	W =  90.000 deg,	P =   0.000 deg,	R =   90.000 deg
};
P[960]{
   GP1:
	UF : 0, UT : 6,		CONFIG : 'N U T, 0, 0, 0',
	X =  -28.903  mm,	Y =   -328.878  mm,	Z =   -247.975  mm,
	W =  90.000 deg,	P =   0.000 deg,	R =   90.000 deg
};
P[961]{
   GP1:
	UF : 0, UT : 6,		CONFIG : 'N U T, 0, 0, 0',
	X =  -30.345  mm,	Y =   -329.747  mm,	Z =   -248.064  mm,
	W =  90.000 deg,	P =   0.000 deg,	R =   90.000 deg
};
P[962]{
   GP1:
	UF : 0, UT : 6,		CONFIG : 'N U T, 0, 0, 0',
	X =  -31.296  mm,	Y =   -330.198  mm,	Z =   -247.828  mm,
	W =  90.000 deg,	P =   0.000 deg,	R =   90.000 deg
};
P[963]{
   GP1:
	UF : 0, UT : 6,		CONFIG : 'N U T, 0, 0, 0',
	X =  -37.082  mm,	Y =   -333.556  mm,	Z =   -247.870  mm,
	W =  90.000 deg,	P =   0.000 deg,	R =   90.000 deg
};
P[964]{
   GP1:
	UF : 0, UT : 6,		CONFIG : 'N U T, 0, 0, 0',
	X =  -38.322  mm,	Y =   -334.338  mm,	Z =   -248.027  mm,
	W =  90.000 deg,	P =   0.000 deg,	R =   90.000 deg
};
P[965]{
   GP1:
	UF : 0, UT : 6,		CONFIG : 'N U T, 0, 0, 0',
	X =  -39.006  mm,	Y =   -334.749  mm,	Z =   -248.069  mm,
	W =  90.000 deg,	P =   0.000 deg,	R =   90.000 deg
};
P[966]{
   GP1:
	UF : 0, UT : 6,		CONFIG : 'N U T, 0, 0, 0',
	X =  -40.131  mm,	Y =   -335.448  mm,	Z =   -248.189  mm,
	W =  90.000 deg,	P =   0.000 deg,	R =   90.000 deg
};
P[967]{
   GP1:
	UF : 0, UT : 6,		CONFIG : 'N U T, 0, 0, 0',
	X =  -41.021  mm,	Y =   -335.924  mm,	Z =   -248.096  mm,
	W =  90.000 deg,	P =   0.000 deg,	R =   90.000 deg
};
P[968]{
   GP1:
	UF : 0, UT : 6,		CONFIG : 'N U T, 0, 0, 0',
	X =  -42.003  mm,	Y =   -336.481  mm,	Z =   -248.073  mm,
	W =  90.000 deg,	P =   0.000 deg,	R =   90.000 deg
};
P[969]{
   GP1:
	UF : 0, UT : 6,		CONFIG : 'N U T, 0, 0, 0',
	X =  -43.049  mm,	Y =   -337.147  mm,	Z =   -248.222  mm,
	W =  90.000 deg,	P =   0.000 deg,	R =   90.000 deg
};
P[970]{
   GP1:
	UF : 0, UT : 6,		CONFIG : 'N U T, 0, 0, 0',
	X =  -43.885  mm,	Y =   -337.634  mm,	Z =   -248.233  mm,
	W =  90.000 deg,	P =   0.000 deg,	R =   90.000 deg
};
P[971]{
   GP1:
	UF : 0, UT : 6,		CONFIG : 'N U T, 0, 0, 0',
	X =  -45.078  mm,	Y =   -338.309  mm,	Z =   -248.202  mm,
	W =  90.000 deg,	P =   0.000 deg,	R =   90.000 deg
};
P[972]{
   GP1:
	UF : 0, UT : 6,		CONFIG : 'N U T, 0, 0, 0',
	X =  -49.857  mm,	Y =   -340.939  mm,	Z =   -247.886  mm,
	W =  90.000 deg,	P =   0.000 deg,	R =   90.000 deg
};
P[973]{
   GP1:
	UF : 0, UT : 6,		CONFIG : 'N U T, 0, 0, 0',
	X =  -51.596  mm,	Y =   -342.068  mm,	Z =   -248.190  mm,
	W =  90.000 deg,	P =   0.000 deg,	R =   90.000 deg
};
P[974]{
   GP1:
	UF : 0, UT : 6,		CONFIG : 'N U T, 0, 0, 0',
	X =  -55.566  mm,	Y =   -344.197  mm,	Z =   -247.792  mm,
	W =  90.000 deg,	P =   0.000 deg,	R =   90.000 deg
};
P[975]{
   GP1:
	UF : 0, UT : 6,		CONFIG : 'N U T, 0, 0, 0',
	X =  -56.702  mm,	Y =   -344.999  mm,	Z =   -248.147  mm,
	W =  90.000 deg,	P =   0.000 deg,	R =   90.000 deg
};
P[976]{
   GP1:
	UF : 0, UT : 6,		CONFIG : 'N U T, 0, 0, 0',
	X =  -58.375  mm,	Y =   -345.890  mm,	Z =   -247.965  mm,
	W =  90.000 deg,	P =   0.000 deg,	R =   90.000 deg
};
P[977]{
   GP1:
	UF : 0, UT : 6,		CONFIG : 'N U T, 0, 0, 0',
	X =  -60.750  mm,	Y =   -347.335  mm,	Z =   -248.145  mm,
	W =  90.000 deg,	P =   0.000 deg,	R =   90.000 deg
};
P[978]{
   GP1:
	UF : 0, UT : 6,		CONFIG : 'N U T, 0, 0, 0',
	X =  -61.386  mm,	Y =   -347.642  mm,	Z =   -247.998  mm,
	W =  90.000 deg,	P =   0.000 deg,	R =   90.000 deg
};
P[979]{
   GP1:
	UF : 0, UT : 6,		CONFIG : 'N U T, 0, 0, 0',
	X =  -63.196  mm,	Y =   -348.624  mm,	Z =   -247.843  mm,
	W =  90.000 deg,	P =   0.000 deg,	R =   90.000 deg
};
P[980]{
   GP1:
	UF : 0, UT : 6,		CONFIG : 'N U T, 0, 0, 0',
	X =  -64.126  mm,	Y =   -349.230  mm,	Z =   -248.010  mm,
	W =  90.000 deg,	P =   0.000 deg,	R =   90.000 deg
};
P[981]{
   GP1:
	UF : 0, UT : 6,		CONFIG : 'N U T, 0, 0, 0',
	X =  -65.042  mm,	Y =   -349.775  mm,	Z =   -248.050  mm,
	W =  90.000 deg,	P =   0.000 deg,	R =   90.000 deg
};
P[982]{
   GP1:
	UF : 0, UT : 6,		CONFIG : 'N U T, 0, 0, 0',
	X =  -68.055  mm,	Y =   -351.565  mm,	Z =   -248.174  mm,
	W =  90.000 deg,	P =   0.000 deg,	R =   90.000 deg
};
P[983]{
   GP1:
	UF : 0, UT : 6,		CONFIG : 'N U T, 0, 0, 0',
	X =  -70.480  mm,	Y =   -352.838  mm,	Z =   -247.864  mm,
	W =  90.000 deg,	P =   0.000 deg,	R =   90.000 deg
};
P[984]{
   GP1:
	UF : 0, UT : 6,		CONFIG : 'N U T, 0, 0, 0',
	X =  -72.242  mm,	Y =   -353.967  mm,	Z =   -248.135  mm,
	W =  90.000 deg,	P =   0.000 deg,	R =   90.000 deg
};
P[985]{
   GP1:
	UF : 0, UT : 6,		CONFIG : 'N U T, 0, 0, 0',
	X =  -73.253  mm,	Y =   -354.525  mm,	Z =   -248.074  mm,
	W =  90.000 deg,	P =   0.000 deg,	R =   90.000 deg
};
P[986]{
   GP1:
	UF : 0, UT : 6,		CONFIG : 'N U T, 0, 0, 0',
	X =  -74.249  mm,	Y =   -355.111  mm,	Z =   -248.099  mm,
	W =  90.000 deg,	P =   0.000 deg,	R =   90.000 deg
};
P[987]{
   GP1:
	UF : 0, UT : 6,		CONFIG : 'N U T, 0, 0, 0',
	X =  -75.340  mm,	Y =   -355.605  mm,	Z =   -247.770  mm,
	W =  90.000 deg,	P =   0.000 deg,	R =   90.000 deg
};
P[988]{
   GP1:
	UF : 0, UT : 6,		CONFIG : 'N U T, 0, 0, 0',
	X =  -77.108  mm,	Y =   -356.686  mm,	Z =   -247.916  mm,
	W =  90.000 deg,	P =   0.000 deg,	R =   90.000 deg
};
P[989]{
   GP1:
	UF : 0, UT : 6,		CONFIG : 'N U T, 0, 0, 0',
	X =  -77.787  mm,	Y =   -357.064  mm,	Z =   -247.884  mm,
	W =  90.000 deg,	P =   0.000 deg,	R =   90.000 deg
};
P[990]{
   GP1:
	UF : 0, UT : 6,		CONFIG : 'N U T, 0, 0, 0',
	X =  -79.134  mm,	Y =   -357.855  mm,	Z =   -247.913  mm,
	W =  90.000 deg,	P =   0.000 deg,	R =   90.000 deg
};
P[991]{
   GP1:
	UF : 0, UT : 6,		CONFIG : 'N U T, 0, 0, 0',
	X =  -81.215  mm,	Y =   -359.115  mm,	Z =   -248.054  mm,
	W =  90.000 deg,	P =   0.000 deg,	R =   90.000 deg
};
P[992]{
   GP1:
	UF : 0, UT : 6,		CONFIG : 'N U T, 0, 0, 0',
	X =  -82.562  mm,	Y =   -359.948  mm,	Z =   -248.191  mm,
	W =  90.000 deg,	P =   0.000 deg,	R =   90.000 deg
};
P[993]{
   GP1:
	UF : 0, UT : 6,		CONFIG : 'N U T, 0, 0, 0',
	X =  -84.553  mm,	Y =   -361.046  mm,	Z =   -248.064  mm,
	W =  90.000 deg,	P =   0.000 deg,	R =   90.000 deg
};
P[994]{
   GP1:
	UF : 0, UT : 6,		CONFIG : 'N U T, 0, 0, 0',
	X =  -85.474  mm,	Y =   -361.519  mm,	Z =   -247.920  mm,
	W =  90.000 deg,	P =   0.000 deg,	R =   90.000 deg
};
P[995]{
   GP1:
	UF : 0, UT : 6,		CONFIG : 'N U T, 0, 0, 0',
	X =  -86.598  mm,	Y =   -362.225  mm,	Z =   -248.060  mm,
	W =  90.000 deg,	P =   0.000 deg,	R =   90.000 deg
};
P[996]{
   GP1:
	UF : 0, UT : 6,		CONFIG : 'N U T, 0, 0, 0',
	X =  -89.940  mm,	Y =   -364.214  mm,	Z =   -248.203  mm,
	W =  90.000 deg,	P =   0.000 deg,	R =   90.000 deg
};
P[997]{
   GP1:
	UF : 0, UT : 6,		CONFIG : 'N U T, 0, 0, 0',
	X =  -90.933  mm,	Y =   -364.603  mm,	Z =   -247.758  mm,
	W =  90.000 deg,	P =   0.000 deg,	R =   90.000 deg
};
P[998]{
   GP1:
	UF : 0, UT : 6,		CONFIG : 'N U T, 0, 0, 0',
	X =  -91.875  mm,	Y =   -365.326  mm,	Z =   -248.193  mm,
	W =  90.000 deg,	P =   0.000 deg,	R =   90.000 deg
};
P[999]{
   GP1:
	UF : 0, UT : 6,		CONFIG : 'N U T, 0, 0, 0',
	X =  -94.257  mm,	Y =   -366.581  mm,	Z =   -247.899  mm,
	W =  90.000 deg,	P =   0.000 deg,	R =   90.000 deg
};
P[1000]{
   GP1:
	UF : 0, UT : 6,		CONFIG : 'N U T, 0, 0, 0',
	X =  -95.224  mm,	Y =   -367.210  mm,	Z =   -248.072  mm,
	W =  90.000 deg,	P =   0.000 deg,	R =   90.000 deg
};
P[1001]{
   GP1:
	UF : 0, UT : 6,		CONFIG : 'N U T, 0, 0, 0',
	X =  -96.301  mm,	Y =   -367.796  mm,	Z =   -247.984  mm,
	W =  90.000 deg,	P =   0.000 deg,	R =   90.000 deg
};
P[1002]{
   GP1:
	UF : 0, UT : 6,		CONFIG : 'N U T, 0, 0, 0',
	X =  -97.537  mm,	Y =   -368.595  mm,	Z =   -248.191  mm,
	W =  90.000 deg,	P =   0.000 deg,	R =   90.000 deg
};
P[1003]{
   GP1:
	UF : 0, UT : 6,		CONFIG : 'N U T, 0, 0, 0',
	X =  -99.221  mm,	Y =   -369.495  mm,	Z =   -248.013  mm,
	W =  90.000 deg,	P =   0.000 deg,	R =   90.000 deg
};
P[1004]{
   GP1:
	UF : 0, UT : 6,		CONFIG : 'N U T, 0, 0, 0',
	X =  -101.503  mm,	Y =   -370.901  mm,	Z =   -248.231  mm,
	W =  90.000 deg,	P =   0.000 deg,	R =   90.000 deg
};
P[1005]{
   GP1:
	UF : 0, UT : 6,		CONFIG : 'N U T, 0, 0, 0',
	X =  -102.830  mm,	Y =   -371.582  mm,	Z =   -248.024  mm,
	W =  90.000 deg,	P =   0.000 deg,	R =   90.000 deg
};
P[1006]{
   GP1:
	UF : 0, UT : 6,		CONFIG : 'N U T, 0, 0, 0',
	X =  -103.563  mm,	Y =   -371.971  mm,	Z =   -247.940  mm,
	W =  90.000 deg,	P =   0.000 deg,	R =   90.000 deg
};
P[1007]{
   GP1:
	UF : 0, UT : 6,		CONFIG : 'N U T, 0, 0, 0',
	X =  -106.169  mm,	Y =   -373.484  mm,	Z =   -247.960  mm,
	W =  90.000 deg,	P =   0.000 deg,	R =   90.000 deg
};
P[1008]{
   GP1:
	UF : 0, UT : 6,		CONFIG : 'N U T, 0, 0, 0',
	X =  -106.807  mm,	Y =   -373.966  mm,	Z =   -248.237  mm,
	W =  90.000 deg,	P =   0.000 deg,	R =   90.000 deg
};
P[1009]{
   GP1:
	UF : 0, UT : 6,		CONFIG : 'N U T, 0, 0, 0',
	X =  -107.493  mm,	Y =   -374.305  mm,	Z =   -248.100  mm,
	W =  90.000 deg,	P =   0.000 deg,	R =   90.000 deg
};
P[1010]{
   GP1:
	UF : 0, UT : 6,		CONFIG : 'N U T, 0, 0, 0',
	X =  -108.733  mm,	Y =   -375.067  mm,	Z =   -248.210  mm,
	W =  90.000 deg,	P =   0.000 deg,	R =   90.000 deg
};
P[1011]{
   GP1:
	UF : 0, UT : 6,		CONFIG : 'N U T, 0, 0, 0',
	X =  -110.528  mm,	Y =   -376.015  mm,	Z =   -247.997  mm,
	W =  90.000 deg,	P =   0.000 deg,	R =   90.000 deg
};
P[1012]{
   GP1:
	UF : 0, UT : 6,		CONFIG : 'N U T, 0, 0, 0',
	X =  -111.099  mm,	Y =   -376.423  mm,	Z =   -248.185  mm,
	W =  90.000 deg,	P =   0.000 deg,	R =   90.000 deg
};
P[1013]{
   GP1:
	UF : 0, UT : 6,		CONFIG : 'N U T, 0, 0, 0',
	X =  -112.870  mm,	Y =   -377.351  mm,	Z =   -247.957  mm,
	W =  90.000 deg,	P =   0.000 deg,	R =   90.000 deg
};
P[1014]{
   GP1:
	UF : 0, UT : 6,		CONFIG : 'N U T, 0, 0, 0',
	X =  -113.558  mm,	Y =   -377.684  mm,	Z =   -247.799  mm,
	W =  90.000 deg,	P =   0.000 deg,	R =   90.000 deg
};
P[1015]{
   GP1:
	UF : 0, UT : 6,		CONFIG : 'N U T, 0, 0, 0',
	X =  -115.265  mm,	Y =   -378.664  mm,	Z =   -247.786  mm,
	W =  90.000 deg,	P =   0.000 deg,	R =   90.000 deg
};
P[1016]{
   GP1:
	UF : 0, UT : 6,		CONFIG : 'N U T, 0, 0, 0',
	X =  -116.104  mm,	Y =   -379.315  mm,	Z =   -248.189  mm,
	W =  90.000 deg,	P =   0.000 deg,	R =   90.000 deg
};
P[1017]{
   GP1:
	UF : 0, UT : 6,		CONFIG : 'N U T, 0, 0, 0',
	X =  -117.677  mm,	Y =   -380.092  mm,	Z =   -247.871  mm,
	W =  90.000 deg,	P =   0.000 deg,	R =   90.000 deg
};
P[1018]{
   GP1:
	UF : 0, UT : 6,		CONFIG : 'N U T, 0, 0, 0',
	X =  -118.616  mm,	Y =   -380.734  mm,	Z =   -248.113  mm,
	W =  90.000 deg,	P =   0.000 deg,	R =   90.000 deg
};
P[1019]{
   GP1:
	UF : 0, UT : 6,		CONFIG : 'N U T, 0, 0, 0',
	X =  -122.113  mm,	Y =   -382.775  mm,	Z =   -248.168  mm,
	W =  90.000 deg,	P =   0.000 deg,	R =   90.000 deg
};
P[1020]{
   GP1:
	UF : 0, UT : 6,		CONFIG : 'N U T, 0, 0, 0',
	X =  -124.559  mm,	Y =   -384.127  mm,	Z =   -248.019  mm,
	W =  90.000 deg,	P =   0.000 deg,	R =   90.000 deg
};
P[1021]{
   GP1:
	UF : 0, UT : 6,		CONFIG : 'N U T, 0, 0, 0',
	X =  -125.422  mm,	Y =   -384.715  mm,	Z =   -248.238  mm,
	W =  90.000 deg,	P =   0.000 deg,	R =   90.000 deg
};
P[1022]{
   GP1:
	UF : 0, UT : 6,		CONFIG : 'N U T, 0, 0, 0',
	X =  -126.709  mm,	Y =   -385.433  mm,	Z =   -248.142  mm,
	W =  90.000 deg,	P =   0.000 deg,	R =   90.000 deg
};
P[1023]{
   GP1:
	UF : 0, UT : 6,		CONFIG : 'N U T, 0, 0, 0',
	X =  -129.563  mm,	Y =   -387.669  mm,	Z =   -248.167  mm,
	W =  90.000 deg,	P =   0.000 deg,	R =   90.000 deg
};
P[1024]{
   GP1:
	UF : 0, UT : 6,		CONFIG : 'N U T, 0, 0, 0',
	X =  -130.198  mm,	Y =   -388.316  mm,	Z =   -248.069  mm,
	W =  90.000 deg,	P =   0.000 deg,	R =   90.000 deg
};
P[1025]{
   GP1:
	UF : 0, UT : 6,		CONFIG : 'N U T, 0, 0, 0',
	X =  -132.423  mm,	Y =   -391.705  mm,	Z =   -248.118  mm,
	W =  90.000 deg,	P =   0.000 deg,	R =   90.000 deg
};
P[1026]{
   GP1:
	UF : 0, UT : 6,		CONFIG : 'N U T, 0, 0, 0',
	X =  -132.726  mm,	Y =   -392.586  mm,	Z =   -248.245  mm,
	W =  90.000 deg,	P =   0.000 deg,	R =   90.000 deg
};
P[1027]{
   GP1:
	UF : 0, UT : 6,		CONFIG : 'N U T, 0, 0, 0',
	X =  -133.115  mm,	Y =   -393.723  mm,	Z =   -248.116  mm,
	W =  90.000 deg,	P =   0.000 deg,	R =   90.000 deg
};
P[1028]{
   GP1:
	UF : 0, UT : 6,		CONFIG : 'N U T, 0, 0, 0',
	X =  -133.602  mm,	Y =   -396.256  mm,	Z =   -247.992  mm,
	W =  90.000 deg,	P =   0.000 deg,	R =   90.000 deg
};
P[1029]{
   GP1:
	UF : 0, UT : 6,		CONFIG : 'N U T, 0, 0, 0',
	X =  -133.574  mm,	Y =   -398.321  mm,	Z =   -248.077  mm,
	W =  90.000 deg,	P =   0.000 deg,	R =   90.000 deg
};
P[1030]{
   GP1:
	UF : 0, UT : 6,		CONFIG : 'N U T, 0, 0, 0',
	X =  -133.207  mm,	Y =   -400.061  mm,	Z =   -248.179  mm,
	W =  90.000 deg,	P =   0.000 deg,	R =   90.000 deg
};
P[1031]{
   GP1:
	UF : 0, UT : 6,		CONFIG : 'N U T, 0, 0, 0',
	X =  -132.889  mm,	Y =   -401.383  mm,	Z =   -248.224  mm,
	W =  90.000 deg,	P =   0.000 deg,	R =   90.000 deg
};
P[1032]{
   GP1:
	UF : 0, UT : 6,		CONFIG : 'N U T, 0, 0, 0',
	X =  -132.012  mm,	Y =   -403.554  mm,	Z =   -248.053  mm,
	W =  90.000 deg,	P =   0.000 deg,	R =   90.000 deg
};
P[1033]{
   GP1:
	UF : 0, UT : 6,		CONFIG : 'N U T, 0, 0, 0',
	X =  -131.322  mm,	Y =   -404.824  mm,	Z =   -248.139  mm,
	W =  90.000 deg,	P =   0.000 deg,	R =   90.000 deg
};
P[1034]{
   GP1:
	UF : 0, UT : 6,		CONFIG : 'N U T, 0, 0, 0',
	X =  -130.983  mm,	Y =   -405.432  mm,	Z =   -248.111  mm,
	W =  90.000 deg,	P =   0.000 deg,	R =   90.000 deg
};
P[1035]{
   GP1:
	UF : 0, UT : 6,		CONFIG : 'N U T, 0, 0, 0',
	X =  -130.285  mm,	Y =   -406.743  mm,	Z =   -247.966  mm,
	W =  90.000 deg,	P =   0.000 deg,	R =   90.000 deg
};
P[1036]{
   GP1:
	UF : 0, UT : 6,		CONFIG : 'N U T, 0, 0, 0',
	X =  -129.882  mm,	Y =   -407.354  mm,	Z =   -248.089  mm,
	W =  90.000 deg,	P =   0.000 deg,	R =   90.000 deg
};
P[1037]{
   GP1:
	UF : 0, UT : 6,		CONFIG : 'N U T, 0, 0, 0',
	X =  -128.584  mm,	Y =   -409.650  mm,	Z =   -248.021  mm,
	W =  90.000 deg,	P =   0.000 deg,	R =   90.000 deg
};
P[1038]{
   GP1:
	UF : 0, UT : 6,		CONFIG : 'N U T, 0, 0, 0',
	X =  -127.392  mm,	Y =   -411.883  mm,	Z =   -247.787  mm,
	W =  90.000 deg,	P =   0.000 deg,	R =   90.000 deg
};
P[1039]{
   GP1:
	UF : 0, UT : 6,		CONFIG : 'N U T, 0, 0, 0',
	X =  -126.637  mm,	Y =   -412.966  mm,	Z =   -248.099  mm,
	W =  90.000 deg,	P =   0.000 deg,	R =   90.000 deg
};
P[1040]{
   GP1:
	UF : 0, UT : 6,		CONFIG : 'N U T, 0, 0, 0',
	X =  -122.435  mm,	Y =   -420.253  mm,	Z =   -248.085  mm,
	W =  90.000 deg,	P =   0.000 deg,	R =   90.000 deg
};
P[1041]{
   GP1:
	UF : 0, UT : 6,		CONFIG : 'N U T, 0, 0, 0',
	X =  -121.804  mm,	Y =   -421.568  mm,	Z =   -247.775  mm,
	W =  90.000 deg,	P =   0.000 deg,	R =   90.000 deg
};
P[1042]{
   GP1:
	UF : 0, UT : 6,		CONFIG : 'N U T, 0, 0, 0',
	X =  -120.774  mm,	Y =   -423.206  mm,	Z =   -247.982  mm,
	W =  90.000 deg,	P =   0.000 deg,	R =   90.000 deg
};
P[1043]{
   GP1:
	UF : 0, UT : 6,		CONFIG : 'N U T, 0, 0, 0',
	X =  -120.097  mm,	Y =   -424.195  mm,	Z =   -248.237  mm,
	W =  90.000 deg,	P =   0.000 deg,	R =   90.000 deg
};
P[1044]{
   GP1:
	UF : 0, UT : 6,		CONFIG : 'N U T, 0, 0, 0',
	X =  -119.414  mm,	Y =   -425.491  mm,	Z =   -248.078  mm,
	W =  90.000 deg,	P =   0.000 deg,	R =   90.000 deg
};
P[1045]{
   GP1:
	UF : 0, UT : 6,		CONFIG : 'N U T, 0, 0, 0',
	X =  -118.894  mm,	Y =   -426.411  mm,	Z =   -248.052  mm,
	W =  90.000 deg,	P =   0.000 deg,	R =   90.000 deg
};
P[1046]{
   GP1:
	UF : 0, UT : 6,		CONFIG : 'N U T, 0, 0, 0',
	X =  -118.256  mm,	Y =   -427.421  mm,	Z =   -248.184  mm,
	W =  90.000 deg,	P =   0.000 deg,	R =   90.000 deg
};
P[1047]{
   GP1:
	UF : 0, UT : 6,		CONFIG : 'N U T, 0, 0, 0',
	X =  -117.760  mm,	Y =   -428.344  mm,	Z =   -248.095  mm,
	W =  90.000 deg,	P =   0.000 deg,	R =   90.000 deg
};
P[1048]{
   GP1:
	UF : 0, UT : 6,		CONFIG : 'N U T, 0, 0, 0',
	X =  -116.499  mm,	Y =   -430.746  mm,	Z =   -247.790  mm,
	W =  90.000 deg,	P =   0.000 deg,	R =   90.000 deg
};
P[1049]{
   GP1:
	UF : 0, UT : 6,		CONFIG : 'N U T, 0, 0, 0',
	X =  -115.798  mm,	Y =   -431.817  mm,	Z =   -247.989  mm,
	W =  90.000 deg,	P =   0.000 deg,	R =   90.000 deg
};
P[1050]{
   GP1:
	UF : 0, UT : 6,		CONFIG : 'N U T, 0, 0, 0',
	X =  -114.795  mm,	Y =   -433.512  mm,	Z =   -248.050  mm,
	W =  90.000 deg,	P =   0.000 deg,	R =   90.000 deg
};
P[1051]{
   GP1:
	UF : 0, UT : 6,		CONFIG : 'N U T, 0, 0, 0',
	X =  -114.179  mm,	Y =   -434.555  mm,	Z =   -248.082  mm,
	W =  90.000 deg,	P =   0.000 deg,	R =   90.000 deg
};
P[1052]{
   GP1:
	UF : 0, UT : 6,		CONFIG : 'N U T, 0, 0, 0',
	X =  -112.942  mm,	Y =   -436.662  mm,	Z =   -248.134  mm,
	W =  90.000 deg,	P =   0.000 deg,	R =   90.000 deg
};
P[1053]{
   GP1:
	UF : 0, UT : 6,		CONFIG : 'N U T, 0, 0, 0',
	X =  -112.334  mm,	Y =   -437.964  mm,	Z =   -247.783  mm,
	W =  90.000 deg,	P =   0.000 deg,	R =   90.000 deg
};
P[1054]{
   GP1:
	UF : 0, UT : 6,		CONFIG : 'N U T, 0, 0, 0',
	X =  -111.595  mm,	Y =   -439.228  mm,	Z =   -247.806  mm,
	W =  90.000 deg,	P =   0.000 deg,	R =   90.000 deg
};
P[1055]{
   GP1:
	UF : 0, UT : 6,		CONFIG : 'N U T, 0, 0, 0',
	X =  -110.365  mm,	Y =   -441.151  mm,	Z =   -248.096  mm,
	W =  90.000 deg,	P =   0.000 deg,	R =   90.000 deg
};
P[1056]{
   GP1:
	UF : 0, UT : 6,		CONFIG : 'N U T, 0, 0, 0',
	X =  -109.824  mm,	Y =   -442.301  mm,	Z =   -247.797  mm,
	W =  90.000 deg,	P =   0.000 deg,	R =   90.000 deg
};
P[1057]{
   GP1:
	UF : 0, UT : 6,		CONFIG : 'N U T, 0, 0, 0',
	X =  -108.955  mm,	Y =   -443.499  mm,	Z =   -248.227  mm,
	W =  90.000 deg,	P =   0.000 deg,	R =   90.000 deg
};
P[1058]{
   GP1:
	UF : 0, UT : 6,		CONFIG : 'N U T, 0, 0, 0',
	X =  -108.580  mm,	Y =   -444.387  mm,	Z =   -247.895  mm,
	W =  90.000 deg,	P =   0.000 deg,	R =   90.000 deg
};
P[1059]{
   GP1:
	UF : 0, UT : 6,		CONFIG : 'N U T, 0, 0, 0',
	X =  -107.695  mm,	Y =   -445.733  mm,	Z =   -248.155  mm,
	W =  90.000 deg,	P =   0.000 deg,	R =   90.000 deg
};
P[1060]{
   GP1:
	UF : 0, UT : 6,		CONFIG : 'N U T, 0, 0, 0',
	X =  -105.502  mm,	Y =   -449.497  mm,	Z =   -248.203  mm,
	W =  90.000 deg,	P =   0.000 deg,	R =   90.000 deg
};
P[1061]{
   GP1:
	UF : 0, UT : 6,		CONFIG : 'N U T, 0, 0, 0',
	X =  -104.845  mm,	Y =   -450.741  mm,	Z =   -248.054  mm,
	W =  90.000 deg,	P =   0.000 deg,	R =   90.000 deg
};
P[1062]{
   GP1:
	UF : 0, UT : 6,		CONFIG : 'N U T, 0, 0, 0',
	X =  -104.462  mm,	Y =   -451.470  mm,	Z =   -247.962  mm,
	W =  90.000 deg,	P =   0.000 deg,	R =   90.000 deg
};
P[1063]{
   GP1:
	UF : 0, UT : 6,		CONFIG : 'N U T, 0, 0, 0',
	X =  -104.089  mm,	Y =   -452.185  mm,	Z =   -247.868  mm,
	W =  90.000 deg,	P =   0.000 deg,	R =   90.000 deg
};
P[1064]{
   GP1:
	UF : 0, UT : 6,		CONFIG : 'N U T, 0, 0, 0',
	X =  -102.684  mm,	Y =   -454.644  mm,	Z =   -247.831  mm,
	W =  90.000 deg,	P =   0.000 deg,	R =   90.000 deg
};
P[1065]{
   GP1:
	UF : 0, UT : 6,		CONFIG : 'N U T, 0, 0, 0',
	X =  -102.091  mm,	Y =   -455.612  mm,	Z =   -247.912  mm,
	W =  90.000 deg,	P =   0.000 deg,	R =   90.000 deg
};
P[1066]{
   GP1:
	UF : 0, UT : 6,		CONFIG : 'N U T, 0, 0, 0',
	X =  -101.461  mm,	Y =   -456.515  mm,	Z =   -248.175  mm,
	W =  90.000 deg,	P =   0.000 deg,	R =   90.000 deg
};
P[1067]{
   GP1:
	UF : 0, UT : 6,		CONFIG : 'N U T, 0, 0, 0',
	X =  -100.753  mm,	Y =   -457.744  mm,	Z =   -248.173  mm,
	W =  90.000 deg,	P =   0.000 deg,	R =   90.000 deg
};
P[1068]{
   GP1:
	UF : 0, UT : 6,		CONFIG : 'N U T, 0, 0, 0',
	X =  -99.853  mm,	Y =   -459.493  mm,	Z =   -247.904  mm,
	W =  90.000 deg,	P =   0.000 deg,	R =   90.000 deg
};
P[1069]{
   GP1:
	UF : 0, UT : 6,		CONFIG : 'N U T, 0, 0, 0',
	X =  -97.147  mm,	Y =   -463.978  mm,	Z =   -248.189  mm,
	W =  90.000 deg,	P =   0.000 deg,	R =   90.000 deg
};
P[1070]{
   GP1:
	UF : 0, UT : 6,		CONFIG : 'N U T, 0, 0, 0',
	X =  -96.488  mm,	Y =   -465.368  mm,	Z =   -247.838  mm,
	W =  90.000 deg,	P =   0.000 deg,	R =   90.000 deg
};
P[1071]{
   GP1:
	UF : 0, UT : 6,		CONFIG : 'N U T, 0, 0, 0',
	X =  -95.821  mm,	Y =   -466.485  mm,	Z =   -247.895  mm,
	W =  90.000 deg,	P =   0.000 deg,	R =   90.000 deg
};
P[1072]{
   GP1:
	UF : 0, UT : 6,		CONFIG : 'N U T, 0, 0, 0',
	X =  -95.262  mm,	Y =   -467.225  mm,	Z =   -248.213  mm,
	W =  90.000 deg,	P =   0.000 deg,	R =   90.000 deg
};
P[1073]{
   GP1:
	UF : 0, UT : 6,		CONFIG : 'N U T, 0, 0, 0',
	X =  -93.623  mm,	Y =   -470.273  mm,	Z =   -247.917  mm,
	W =  90.000 deg,	P =   0.000 deg,	R =   90.000 deg
};
P[1074]{
   GP1:
	UF : 0, UT : 6,		CONFIG : 'N U T, 0, 0, 0',
	X =  -92.822  mm,	Y =   -471.615  mm,	Z =   -247.983  mm,
	W =  90.000 deg,	P =   0.000 deg,	R =   90.000 deg
};
P[1075]{
   GP1:
	UF : 0, UT : 6,		CONFIG : 'N U T, 0, 0, 0',
	X =  -92.155  mm,	Y =   -472.636  mm,	Z =   -248.172  mm,
	W =  90.000 deg,	P =   0.000 deg,	R =   90.000 deg
};
P[1076]{
   GP1:
	UF : 0, UT : 6,		CONFIG : 'N U T, 0, 0, 0',
	X =  -91.150  mm,	Y =   -474.438  mm,	Z =   -248.086  mm,
	W =  90.000 deg,	P =   0.000 deg,	R =   90.000 deg
};
P[1077]{
   GP1:
	UF : 0, UT : 6,		CONFIG : 'N U T, 0, 0, 0',
	X =  -90.497  mm,	Y =   -475.686  mm,	Z =   -247.922  mm,
	W =  90.000 deg,	P =   0.000 deg,	R =   90.000 deg
};
P[1078]{
   GP1:
	UF : 0, UT : 6,		CONFIG : 'N U T, 0, 0, 0',
	X =  -88.747  mm,	Y =   -478.722  mm,	Z =   -247.912  mm,
	W =  90.000 deg,	P =   0.000 deg,	R =   90.000 deg
};
P[1079]{
   GP1:
	UF : 0, UT : 6,		CONFIG : 'N U T, 0, 0, 0',
	X =  -88.249  mm,	Y =   -479.554  mm,	Z =   -247.957  mm,
	W =  90.000 deg,	P =   0.000 deg,	R =   90.000 deg
};
P[1080]{
   GP1:
	UF : 0, UT : 6,		CONFIG : 'N U T, 0, 0, 0',
	X =  -87.020  mm,	Y =   -481.678  mm,	Z =   -247.963  mm,
	W =  90.000 deg,	P =   0.000 deg,	R =   90.000 deg
};
P[1081]{
   GP1:
	UF : 0, UT : 6,		CONFIG : 'N U T, 0, 0, 0',
	X =  -86.491  mm,	Y =   -482.557  mm,	Z =   -248.017  mm,
	W =  90.000 deg,	P =   0.000 deg,	R =   90.000 deg
};
P[1082]{
   GP1:
	UF : 0, UT : 6,		CONFIG : 'N U T, 0, 0, 0',
	X =  -83.260  mm,	Y =   -488.237  mm,	Z =   -247.897  mm,
	W =  90.000 deg,	P =   0.000 deg,	R =   90.000 deg
};
P[1083]{
   GP1:
	UF : 0, UT : 6,		CONFIG : 'N U T, 0, 0, 0',
	X =  -81.554  mm,	Y =   -491.053  mm,	Z =   -248.092  mm,
	W =  90.000 deg,	P =   0.000 deg,	R =   90.000 deg
};
P[1084]{
   GP1:
	UF : 0, UT : 6,		CONFIG : 'N U T, 0, 0, 0',
	X =  -79.066  mm,	Y =   -495.264  mm,	Z =   -248.227  mm,
	W =  90.000 deg,	P =   0.000 deg,	R =   90.000 deg
};
P[1085]{
   GP1:
	UF : 0, UT : 6,		CONFIG : 'N U T, 0, 0, 0',
	X =  -78.745  mm,	Y =   -496.131  mm,	Z =   -247.793  mm,
	W =  90.000 deg,	P =   0.000 deg,	R =   90.000 deg
};
P[1086]{
   GP1:
	UF : 0, UT : 6,		CONFIG : 'N U T, 0, 0, 0',
	X =  -76.359  mm,	Y =   -499.951  mm,	Z =   -248.231  mm,
	W =  90.000 deg,	P =   0.000 deg,	R =   90.000 deg
};
P[1087]{
   GP1:
	UF : 0, UT : 6,		CONFIG : 'N U T, 0, 0, 0',
	X =  -75.085  mm,	Y =   -502.217  mm,	Z =   -248.147  mm,
	W =  90.000 deg,	P =   0.000 deg,	R =   90.000 deg
};
P[1088]{
   GP1:
	UF : 0, UT : 6,		CONFIG : 'N U T, 0, 0, 0',
	X =  -74.296  mm,	Y =   -503.735  mm,	Z =   -247.934  mm,
	W =  90.000 deg,	P =   0.000 deg,	R =   90.000 deg
};
P[1089]{
   GP1:
	UF : 0, UT : 6,		CONFIG : 'N U T, 0, 0, 0',
	X =  -73.716  mm,	Y =   -504.717  mm,	Z =   -247.965  mm,
	W =  90.000 deg,	P =   0.000 deg,	R =   90.000 deg
};
P[1090]{
   GP1:
	UF : 0, UT : 6,		CONFIG : 'N U T, 0, 0, 0',
	X =  -73.101  mm,	Y =   -505.743  mm,	Z =   -248.019  mm,
	W =  90.000 deg,	P =   0.000 deg,	R =   90.000 deg
};
P[1091]{
   GP1:
	UF : 0, UT : 6,		CONFIG : 'N U T, 0, 0, 0',
	X =  -72.668  mm,	Y =   -506.616  mm,	Z =   -247.847  mm,
	W =  90.000 deg,	P =   0.000 deg,	R =   90.000 deg
};
P[1092]{
   GP1:
	UF : 0, UT : 6,		CONFIG : 'N U T, 0, 0, 0',
	X =  -71.102  mm,	Y =   -509.080  mm,	Z =   -248.194  mm,
	W =  90.000 deg,	P =   0.000 deg,	R =   90.000 deg
};
P[1093]{
   GP1:
	UF : 0, UT : 6,		CONFIG : 'N U T, 0, 0, 0',
	X =  -69.772  mm,	Y =   -511.607  mm,	Z =   -247.882  mm,
	W =  90.000 deg,	P =   0.000 deg,	R =   90.000 deg
};
P[1094]{
   GP1:
	UF : 0, UT : 6,		CONFIG : 'N U T, 0, 0, 0',
	X =  -68.834  mm,	Y =   -513.104  mm,	Z =   -248.060  mm,
	W =  90.000 deg,	P =   0.000 deg,	R =   90.000 deg
};
P[1095]{
   GP1:
	UF : 0, UT : 6,		CONFIG : 'N U T, 0, 0, 0',
	X =  -68.421  mm,	Y =   -513.798  mm,	Z =   -248.091  mm,
	W =  90.000 deg,	P =   0.000 deg,	R =   90.000 deg
};
P[1096]{
   GP1:
	UF : 0, UT : 6,		CONFIG : 'N U T, 0, 0, 0',
	X =  -67.867  mm,	Y =   -514.903  mm,	Z =   -247.889  mm,
	W =  90.000 deg,	P =   0.000 deg,	R =   90.000 deg
};
P[1097]{
   GP1:
	UF : 0, UT : 6,		CONFIG : 'N U T, 0, 0, 0',
	X =  -67.447  mm,	Y =   -515.576  mm,	Z =   -247.964  mm,
	W =  90.000 deg,	P =   0.000 deg,	R =   90.000 deg
};
P[1098]{
   GP1:
	UF : 0, UT : 6,		CONFIG : 'N U T, 0, 0, 0',
	X =  -65.365  mm,	Y =   -519.077  mm,	Z =   -248.110  mm,
	W =  90.000 deg,	P =   0.000 deg,	R =   90.000 deg
};
P[1099]{
   GP1:
	UF : 0, UT : 6,		CONFIG : 'N U T, 0, 0, 0',
	X =  -64.641  mm,	Y =   -520.439  mm,	Z =   -247.960  mm,
	W =  90.000 deg,	P =   0.000 deg,	R =   90.000 deg
};
P[1100]{
   GP1:
	UF : 0, UT : 6,		CONFIG : 'N U T, 0, 0, 0',
	X =  -63.019  mm,	Y =   -523.252  mm,	Z =   -247.954  mm,
	W =  90.000 deg,	P =   0.000 deg,	R =   90.000 deg
};
P[1101]{
   GP1:
	UF : 0, UT : 6,		CONFIG : 'N U T, 0, 0, 0',
	X =  -61.572  mm,	Y =   -525.772  mm,	Z =   -247.935  mm,
	W =  90.000 deg,	P =   0.000 deg,	R =   90.000 deg
};
P[1102]{
   GP1:
	UF : 0, UT : 6,		CONFIG : 'N U T, 0, 0, 0',
	X =  -57.398  mm,	Y =   -532.795  mm,	Z =   -248.222  mm,
	W =  90.000 deg,	P =   0.000 deg,	R =   90.000 deg
};
P[1103]{
   GP1:
	UF : 0, UT : 6,		CONFIG : 'N U T, 0, 0, 0',
	X =  -56.956  mm,	Y =   -533.648  mm,	Z =   -248.101  mm,
	W =  90.000 deg,	P =   0.000 deg,	R =   90.000 deg
};
P[1104]{
   GP1:
	UF : 0, UT : 6,		CONFIG : 'N U T, 0, 0, 0',
	X =  -53.366  mm,	Y =   -539.846  mm,	Z =   -248.130  mm,
	W =  90.000 deg,	P =   0.000 deg,	R =   90.000 deg
};
P[1105]{
   GP1:
	UF : 0, UT : 6,		CONFIG : 'N U T, 0, 0, 0',
	X =  -52.923  mm,	Y =   -540.786  mm,	Z =   -247.884  mm,
	W =  90.000 deg,	P =   0.000 deg,	R =   90.000 deg
};
P[1106]{
   GP1:
	UF : 0, UT : 6,		CONFIG : 'N U T, 0, 0, 0',
	X =  -52.193  mm,	Y =   -542.081  mm,	Z =   -247.845  mm,
	W =  90.000 deg,	P =   0.000 deg,	R =   90.000 deg
};
P[1107]{
   GP1:
	UF : 0, UT : 6,		CONFIG : 'N U T, 0, 0, 0',
	X =  -50.214  mm,	Y =   -545.475  mm,	Z =   -247.891  mm,
	W =  90.000 deg,	P =   0.000 deg,	R =   90.000 deg
};
P[1108]{
   GP1:
	UF : 0, UT : 6,		CONFIG : 'N U T, 0, 0, 0',
	X =  -49.708  mm,	Y =   -546.190  mm,	Z =   -248.114  mm,
	W =  90.000 deg,	P =   0.000 deg,	R =   90.000 deg
};
P[1109]{
   GP1:
	UF : 0, UT : 6,		CONFIG : 'N U T, 0, 0, 0',
	X =  -49.193  mm,	Y =   -547.125  mm,	Z =   -248.057  mm,
	W =  90.000 deg,	P =   0.000 deg,	R =   90.000 deg
};
P[1110]{
   GP1:
	UF : 0, UT : 6,		CONFIG : 'N U T, 0, 0, 0',
	X =  -48.234  mm,	Y =   -548.642  mm,	Z =   -248.257  mm,
	W =  90.000 deg,	P =   0.000 deg,	R =   90.000 deg
};
P[1111]{
   GP1:
	UF : 0, UT : 6,		CONFIG : 'N U T, 0, 0, 0',
	X =  -47.825  mm,	Y =   -549.680  mm,	Z =   -247.794  mm,
	W =  90.000 deg,	P =   0.000 deg,	R =   90.000 deg
};
P[1112]{
   GP1:
	UF : 0, UT : 6,		CONFIG : 'N U T, 0, 0, 0',
	X =  -46.805  mm,	Y =   -551.289  mm,	Z =   -248.017  mm,
	W =  90.000 deg,	P =   0.000 deg,	R =   90.000 deg
};
P[1113]{
   GP1:
	UF : 0, UT : 6,		CONFIG : 'N U T, 0, 0, 0',
	X =  -46.223  mm,	Y =   -552.271  mm,	Z =   -248.052  mm,
	W =  90.000 deg,	P =   0.000 deg,	R =   90.000 deg
};
P[1114]{
   GP1:
	UF : 0, UT : 6,		CONFIG : 'N U T, 0, 0, 0',
	X =  -44.506  mm,	Y =   -555.413  mm,	Z =   -247.819  mm,
	W =  90.000 deg,	P =   0.000 deg,	R =   90.000 deg
};
P[1115]{
   GP1:
	UF : 0, UT : 6,		CONFIG : 'N U T, 0, 0, 0',
	X =  -43.578  mm,	Y =   -556.840  mm,	Z =   -248.070  mm,
	W =  90.000 deg,	P =   0.000 deg,	R =   90.000 deg
};
P[1116]{
   GP1:
	UF : 0, UT : 6,		CONFIG : 'N U T, 0, 0, 0',
	X =  -42.948  mm,	Y =   -558.034  mm,	Z =   -247.928  mm,
	W =  90.000 deg,	P =   0.000 deg,	R =   90.000 deg
};
P[1117]{
   GP1:
	UF : 0, UT : 6,		CONFIG : 'N U T, 0, 0, 0',
	X =  -42.308  mm,	Y =   -559.005  mm,	Z =   -248.118  mm,
	W =  90.000 deg,	P =   0.000 deg,	R =   90.000 deg
};
P[1118]{
   GP1:
	UF : 0, UT : 6,		CONFIG : 'N U T, 0, 0, 0',
	X =  -41.829  mm,	Y =   -559.923  mm,	Z =   -247.992  mm,
	W =  90.000 deg,	P =   0.000 deg,	R =   90.000 deg
};
P[1119]{
   GP1:
	UF : 0, UT : 6,		CONFIG : 'N U T, 0, 0, 0',
	X =  -40.904  mm,	Y =   -561.498  mm,	Z =   -248.032  mm,
	W =  90.000 deg,	P =   0.000 deg,	R =   90.000 deg
};
P[1120]{
   GP1:
	UF : 0, UT : 6,		CONFIG : 'N U T, 0, 0, 0',
	X =  -39.521  mm,	Y =   -564.018  mm,	Z =   -247.859  mm,
	W =  90.000 deg,	P =   0.000 deg,	R =   90.000 deg
};
P[1121]{
   GP1:
	UF : 0, UT : 6,		CONFIG : 'N U T, 0, 0, 0',
	X =  -39.057  mm,	Y =   -564.604  mm,	Z =   -248.162  mm,
	W =  90.000 deg,	P =   0.000 deg,	R =   90.000 deg
};
P[1122]{
   GP1:
	UF : 0, UT : 6,		CONFIG : 'N U T, 0, 0, 0',
	X =  -38.696  mm,	Y =   -565.396  mm,	Z =   -247.930  mm,
	W =  90.000 deg,	P =   0.000 deg,	R =   90.000 deg
};
P[1123]{
   GP1:
	UF : 0, UT : 6,		CONFIG : 'N U T, 0, 0, 0',
	X =  -37.832  mm,	Y =   -566.741  mm,	Z =   -248.141  mm,
	W =  90.000 deg,	P =   0.000 deg,	R =   90.000 deg
};
P[1124]{
   GP1:
	UF : 0, UT : 6,		CONFIG : 'N U T, 0, 0, 0',
	X =  -32.699  mm,	Y =   -575.894  mm,	Z =   -247.770  mm,
	W =  90.000 deg,	P =   0.000 deg,	R =   90.000 deg
};
P[1125]{
   GP1:
	UF : 0, UT : 6,		CONFIG : 'N U T, 0, 0, 0',
	X =  -31.483  mm,	Y =   -577.930  mm,	Z =   -247.868  mm,
	W =  90.000 deg,	P =   0.000 deg,	R =   90.000 deg
};
P[1126]{
   GP1:
	UF : 0, UT : 6,		CONFIG : 'N U T, 0, 0, 0',
	X =  -31.139  mm,	Y =   -578.605  mm,	Z =   -247.759  mm,
	W =  90.000 deg,	P =   0.000 deg,	R =   90.000 deg
};
P[1127]{
   GP1:
	UF : 0, UT : 6,		CONFIG : 'N U T, 0, 0, 0',
	X =  -30.752  mm,	Y =   -578.956  mm,	Z =   -248.207  mm,
	W =  90.000 deg,	P =   0.000 deg,	R =   90.000 deg
};
P[1128]{
   GP1:
	UF : 0, UT : 6,		CONFIG : 'N U T, 0, 0, 0',
	X =  -30.298  mm,	Y =   -579.876  mm,	Z =   -248.019  mm,
	W =  90.000 deg,	P =   0.000 deg,	R =   90.000 deg
};
P[1129]{
   GP1:
	UF : 0, UT : 6,		CONFIG : 'N U T, 0, 0, 0',
	X =  -29.990  mm,	Y =   -580.575  mm,	Z =   -247.786  mm,
	W =  90.000 deg,	P =   0.000 deg,	R =   90.000 deg
};
P[1130]{
   GP1:
	UF : 0, UT : 6,		CONFIG : 'N U T, 0, 0, 0',
	X =  -29.187  mm,	Y =   -581.930  mm,	Z =   -247.837  mm,
	W =  90.000 deg,	P =   0.000 deg,	R =   90.000 deg
};
P[1131]{
   GP1:
	UF : 0, UT : 6,		CONFIG : 'N U T, 0, 0, 0',
	X =  -28.674  mm,	Y =   -582.529  mm,	Z =   -248.241  mm,
	W =  90.000 deg,	P =   0.000 deg,	R =   90.000 deg
};
P[1132]{
   GP1:
	UF : 0, UT : 6,		CONFIG : 'N U T, 0, 0, 0',
	X =  -27.965  mm,	Y =   -583.864  mm,	Z =   -248.091  mm,
	W =  90.000 deg,	P =   0.000 deg,	R =   90.000 deg
};
P[1133]{
   GP1:
	UF : 0, UT : 6,		CONFIG : 'N U T, 0, 0, 0',
	X =  -27.188  mm,	Y =   -585.203  mm,	Z =   -248.102  mm,
	W =  90.000 deg,	P =   0.000 deg,	R =   90.000 deg
};
P[1134]{
   GP1:
	UF : 0, UT : 6,		CONFIG : 'N U T, 0, 0, 0',
	X =  -26.153  mm,	Y =   -587.031  mm,	Z =   -248.054  mm,
	W =  90.000 deg,	P =   0.000 deg,	R =   90.000 deg
};
P[1135]{
   GP1:
	UF : 0, UT : 6,		CONFIG : 'N U T, 0, 0, 0',
	X =  -24.347  mm,	Y =   -590.327  mm,	Z =   -247.816  mm,
	W =  90.000 deg,	P =   0.000 deg,	R =   90.000 deg
};
P[1136]{
   GP1:
	UF : 0, UT : 6,		CONFIG : 'N U T, 0, 0, 0',
	X =  -23.297  mm,	Y =   -592.095  mm,	Z =   -247.889  mm,
	W =  90.000 deg,	P =   0.000 deg,	R =   90.000 deg
};
P[1137]{
   GP1:
	UF : 0, UT : 6,		CONFIG : 'N U T, 0, 0, 0',
	X =  -22.300  mm,	Y =   -593.661  mm,	Z =   -248.115  mm,
	W =  90.000 deg,	P =   0.000 deg,	R =   90.000 deg
};
P[1138]{
   GP1:
	UF : 0, UT : 6,		CONFIG : 'N U T, 0, 0, 0',
	X =  -20.918  mm,	Y =   -596.069  mm,	Z =   -248.095  mm,
	W =  90.000 deg,	P =   0.000 deg,	R =   90.000 deg
};
P[1139]{
   GP1:
	UF : 0, UT : 6,		CONFIG : 'N U T, 0, 0, 0',
	X =  -20.531  mm,	Y =   -596.837  mm,	Z =   -247.958  mm,
	W =  90.000 deg,	P =   0.000 deg,	R =   90.000 deg
};
P[1140]{
   GP1:
	UF : 0, UT : 6,		CONFIG : 'N U T, 0, 0, 0',
	X =  -20.072  mm,	Y =   -597.758  mm,	Z =   -247.779  mm,
	W =  90.000 deg,	P =   0.000 deg,	R =   90.000 deg
};
P[1141]{
   GP1:
	UF : 0, UT : 6,		CONFIG : 'N U T, 0, 0, 0',
	X =  -19.608  mm,	Y =   -598.514  mm,	Z =   -247.847  mm,
	W =  90.000 deg,	P =   0.000 deg,	R =   90.000 deg
};
P[1142]{
   GP1:
	UF : 0, UT : 6,		CONFIG : 'N U T, 0, 0, 0',
	X =  -18.986  mm,	Y =   -599.449  mm,	Z =   -248.045  mm,
	W =  90.000 deg,	P =   0.000 deg,	R =   90.000 deg
};
P[1143]{
   GP1:
	UF : 0, UT : 6,		CONFIG : 'N U T, 0, 0, 0',
	X =  -18.637  mm,	Y =   -600.169  mm,	Z =   -247.883  mm,
	W =  90.000 deg,	P =   0.000 deg,	R =   90.000 deg
};
P[1144]{
   GP1:
	UF : 0, UT : 6,		CONFIG : 'N U T, 0, 0, 0',
	X =  -17.727  mm,	Y =   -601.597  mm,	Z =   -248.093  mm,
	W =  90.000 deg,	P =   0.000 deg,	R =   90.000 deg
};
P[1145]{
   GP1:
	UF : 0, UT : 6,		CONFIG : 'N U T, 0, 0, 0',
	X =  -16.284  mm,	Y =   -604.191  mm,	Z =   -247.958  mm,
	W =  90.000 deg,	P =   0.000 deg,	R =   90.000 deg
};
P[1146]{
   GP1:
	UF : 0, UT : 6,		CONFIG : 'N U T, 0, 0, 0',
	X =  -14.346  mm,	Y =   -607.379  mm,	Z =   -248.193  mm,
	W =  90.000 deg,	P =   0.000 deg,	R =   90.000 deg
};
P[1147]{
   GP1:
	UF : 0, UT : 6,		CONFIG : 'N U T, 0, 0, 0',
	X =  -13.559  mm,	Y =   -608.835  mm,	Z =   -248.063  mm,
	W =  90.000 deg,	P =   0.000 deg,	R =   90.000 deg
};
P[1148]{
   GP1:
	UF : 0, UT : 6,		CONFIG : 'N U T, 0, 0, 0',
	X =  -12.053  mm,	Y =   -611.530  mm,	Z =   -247.942  mm,
	W =  90.000 deg,	P =   0.000 deg,	R =   90.000 deg
};
P[1149]{
   GP1:
	UF : 0, UT : 6,		CONFIG : 'N U T, 0, 0, 0',
	X =  -11.282  mm,	Y =   -612.784  mm,	Z =   -248.056  mm,
	W =  90.000 deg,	P =   0.000 deg,	R =   90.000 deg
};
P[1150]{
   GP1:
	UF : 0, UT : 6,		CONFIG : 'N U T, 0, 0, 0',
	X =  -10.510  mm,	Y =   -614.028  mm,	Z =   -248.186  mm,
	W =  90.000 deg,	P =   0.000 deg,	R =   90.000 deg
};
P[1151]{
   GP1:
	UF : 0, UT : 6,		CONFIG : 'N U T, 0, 0, 0',
	X =  -9.980  mm,	Y =   -614.941  mm,	Z =   -248.192  mm,
	W =  90.000 deg,	P =   0.000 deg,	R =   90.000 deg
};
P[1152]{
   GP1:
	UF : 0, UT : 6,		CONFIG : 'N U T, 0, 0, 0',
	X =  -9.685  mm,	Y =   -615.737  mm,	Z =   -247.795  mm,
	W =  90.000 deg,	P =   0.000 deg,	R =   90.000 deg
};
P[1153]{
   GP1:
	UF : 0, UT : 6,		CONFIG : 'N U T, 0, 0, 0',
	X =  -8.057  mm,	Y =   -618.300  mm,	Z =   -248.153  mm,
	W =  90.000 deg,	P =   0.000 deg,	R =   90.000 deg
};
P[1154]{
   GP1:
	UF : 0, UT : 6,		CONFIG : 'N U T, 0, 0, 0',
	X =  -7.754  mm,	Y =   -618.926  mm,	Z =   -248.012  mm,
	W =  90.000 deg,	P =   0.000 deg,	R =   90.000 deg
};
P[1155]{
   GP1:
	UF : 0, UT : 6,		CONFIG : 'N U T, 0, 0, 0',
	X =  -6.085  mm,	Y =   -621.714  mm,	Z =   -248.153  mm,
	W =  90.000 deg,	P =   0.000 deg,	R =   90.000 deg
};
P[1156]{
   GP1:
	UF : 0, UT : 6,		CONFIG : 'N U T, 0, 0, 0',
	X =  -5.770  mm,	Y =   -622.460  mm,	Z =   -247.874  mm,
	W =  90.000 deg,	P =   0.000 deg,	R =   90.000 deg
};
P[1157]{
   GP1:
	UF : 0, UT : 6,		CONFIG : 'N U T, 0, 0, 0',
	X =  -5.428  mm,	Y =   -623.057  mm,	Z =   -247.870  mm,
	W =  90.000 deg,	P =   0.000 deg,	R =   90.000 deg
};
P[1158]{
   GP1:
	UF : 0, UT : 6,		CONFIG : 'N U T, 0, 0, 0',
	X =  -4.239  mm,	Y =   -625.010  mm,	Z =   -248.016  mm,
	W =  90.000 deg,	P =   0.000 deg,	R =   90.000 deg
};
P[1159]{
   GP1:
	UF : 0, UT : 6,		CONFIG : 'N U T, 0, 0, 0',
	X =  -3.634  mm,	Y =   -626.063  mm,	Z =   -248.008  mm,
	W =  90.000 deg,	P =   0.000 deg,	R =   90.000 deg
};
P[1160]{
   GP1:
	UF : 0, UT : 6,		CONFIG : 'N U T, 0, 0, 0',
	X =  -3.108  mm,	Y =   -626.975  mm,	Z =   -248.008  mm,
	W =  90.000 deg,	P =   0.000 deg,	R =   90.000 deg
};
P[1161]{
   GP1:
	UF : 0, UT : 6,		CONFIG : 'N U T, 0, 0, 0',
	X =  -2.670  mm,	Y =   -627.703  mm,	Z =   -248.050  mm,
	W =  90.000 deg,	P =   0.000 deg,	R =   90.000 deg
};
P[1162]{
   GP1:
	UF : 0, UT : 6,		CONFIG : 'N U T, 0, 0, 0',
	X =  0.997  mm,	Y =   -634.188  mm,	Z =   -247.865  mm,
	W =  90.000 deg,	P =   0.000 deg,	R =   90.000 deg
};
P[1163]{
   GP1:
	UF : 0, UT : 6,		CONFIG : 'N U T, 0, 0, 0',
	X =  1.751  mm,	Y =   -635.415  mm,	Z =   -247.973  mm,
	W =  90.000 deg,	P =   0.000 deg,	R =   90.000 deg
};
P[1164]{
   GP1:
	UF : 0, UT : 6,		CONFIG : 'N U T, 0, 0, 0',
	X =  2.702  mm,	Y =   -637.011  mm,	Z =   -248.046  mm,
	W =  90.000 deg,	P =   0.000 deg,	R =   90.000 deg
};
P[1165]{
   GP1:
	UF : 0, UT : 6,		CONFIG : 'N U T, 0, 0, 0',
	X =  3.634  mm,	Y =   -638.520  mm,	Z =   -248.192  mm,
	W =  90.000 deg,	P =   0.000 deg,	R =   90.000 deg
};
P[1166]{
   GP1:
	UF : 0, UT : 6,		CONFIG : 'N U T, 0, 0, 0',
	X =  4.021  mm,	Y =   -639.344  mm,	Z =   -247.976  mm,
	W =  90.000 deg,	P =   0.000 deg,	R =   90.000 deg
};
P[1167]{
   GP1:
	UF : 0, UT : 6,		CONFIG : 'N U T, 0, 0, 0',
	X =  4.368  mm,	Y =   -639.942  mm,	Z =   -247.983  mm,
	W =  90.000 deg,	P =   0.000 deg,	R =   90.000 deg
};
P[1168]{
   GP1:
	UF : 0, UT : 6,		CONFIG : 'N U T, 0, 0, 0',
	X =  5.071  mm,	Y =   -641.138  mm,	Z =   -248.012  mm,
	W =  90.000 deg,	P =   0.000 deg,	R =   90.000 deg
};
P[1169]{
   GP1:
	UF : 0, UT : 6,		CONFIG : 'N U T, 0, 0, 0',
	X =  6.511  mm,	Y =   -643.683  mm,	Z =   -247.939  mm,
	W =  90.000 deg,	P =   0.000 deg,	R =   90.000 deg
};
P[1170]{
   GP1:
	UF : 0, UT : 6,		CONFIG : 'N U T, 0, 0, 0',
	X =  6.987  mm,	Y =   -644.578  mm,	Z =   -247.843  mm,
	W =  90.000 deg,	P =   0.000 deg,	R =   90.000 deg
};
P[1171]{
   GP1:
	UF : 0, UT : 6,		CONFIG : 'N U T, 0, 0, 0',
	X =  7.409  mm,	Y =   -645.311  mm,	Z =   -247.839  mm,
	W =  90.000 deg,	P =   0.000 deg,	R =   90.000 deg
};
P[1172]{
   GP1:
	UF : 0, UT : 6,		CONFIG : 'N U T, 0, 0, 0',
	X =  7.999  mm,	Y =   -646.275  mm,	Z =   -247.919  mm,
	W =  90.000 deg,	P =   0.000 deg,	R =   90.000 deg
};
P[1173]{
   GP1:
	UF : 0, UT : 6,		CONFIG : 'N U T, 0, 0, 0',
	X =  8.748  mm,	Y =   -647.589  mm,	Z =   -247.892  mm,
	W =  90.000 deg,	P =   0.000 deg,	R =   90.000 deg
};
P[1174]{
   GP1:
	UF : 0, UT : 6,		CONFIG : 'N U T, 0, 0, 0',
	X =  9.520  mm,	Y =   -648.972  mm,	Z =   -247.830  mm,
	W =  90.000 deg,	P =   0.000 deg,	R =   90.000 deg
};
P[1175]{
   GP1:
	UF : 0, UT : 6,		CONFIG : 'N U T, 0, 0, 0',
	X =  9.891  mm,	Y =   -649.630  mm,	Z =   -247.810  mm,
	W =  90.000 deg,	P =   0.000 deg,	R =   90.000 deg
};
P[1176]{
   GP1:
	UF : 0, UT : 6,		CONFIG : 'N U T, 0, 0, 0',
	X =  10.256  mm,	Y =   -650.287  mm,	Z =   -247.776  mm,
	W =  90.000 deg,	P =   0.000 deg,	R =   90.000 deg
};
P[1177]{
   GP1:
	UF : 0, UT : 6,		CONFIG : 'N U T, 0, 0, 0',
	X =  11.208  mm,	Y =   -651.861  mm,	Z =   -247.879  mm,
	W =  90.000 deg,	P =   0.000 deg,	R =   90.000 deg
};
P[1178]{
   GP1:
	UF : 0, UT : 6,		CONFIG : 'N U T, 0, 0, 0',
	X =  12.424  mm,	Y =   -653.767  mm,	Z =   -248.159  mm,
	W =  90.000 deg,	P =   0.000 deg,	R =   90.000 deg
};
P[1179]{
   GP1:
	UF : 0, UT : 6,		CONFIG : 'N U T, 0, 0, 0',
	X =  13.304  mm,	Y =   -655.482  mm,	Z =   -247.893  mm,
	W =  90.000 deg,	P =   0.000 deg,	R =   90.000 deg
};
P[1180]{
   GP1:
	UF : 0, UT : 6,		CONFIG : 'N U T, 0, 0, 0',
	X =  14.169  mm,	Y =   -656.928  mm,	Z =   -247.966  mm,
	W =  90.000 deg,	P =   0.000 deg,	R =   90.000 deg
};
P[1181]{
   GP1:
	UF : 0, UT : 6,		CONFIG : 'N U T, 0, 0, 0',
	X =  15.058  mm,	Y =   -658.394  mm,	Z =   -248.068  mm,
	W =  90.000 deg,	P =   0.000 deg,	R =   90.000 deg
};
P[1182]{
   GP1:
	UF : 0, UT : 6,		CONFIG : 'N U T, 0, 0, 0',
	X =  16.118  mm,	Y =   -660.429  mm,	Z =   -247.789  mm,
	W =  90.000 deg,	P =   0.000 deg,	R =   90.000 deg
};
P[1183]{
   GP1:
	UF : 0, UT : 6,		CONFIG : 'N U T, 0, 0, 0',
	X =  17.827  mm,	Y =   -663.376  mm,	Z =   -247.807  mm,
	W =  90.000 deg,	P =   0.000 deg,	R =   90.000 deg
};
P[1184]{
   GP1:
	UF : 0, UT : 6,		CONFIG : 'N U T, 0, 0, 0',
	X =  18.698  mm,	Y =   -664.612  mm,	Z =   -248.190  mm,
	W =  90.000 deg,	P =   0.000 deg,	R =   90.000 deg
};
P[1185]{
   GP1:
	UF : 0, UT : 6,		CONFIG : 'N U T, 0, 0, 0',
	X =  21.077  mm,	Y =   -668.938  mm,	Z =   -247.901  mm,
	W =  90.000 deg,	P =   0.000 deg,	R =   90.000 deg
};
P[1186]{
   GP1:
	UF : 0, UT : 6,		CONFIG : 'N U T, 0, 0, 0',
	X =  21.630  mm,	Y =   -669.698  mm,	Z =   -248.179  mm,
	W =  90.000 deg,	P =   0.000 deg,	R =   90.000 deg
};
P[1187]{
   GP1:
	UF : 0, UT : 6,		CONFIG : 'N U T, 0, 0, 0',
	X =  22.787  mm,	Y =   -671.709  mm,	Z =   -248.170  mm,
	W =  90.000 deg,	P =   0.000 deg,	R =   90.000 deg
};
P[1188]{
   GP1:
	UF : 0, UT : 6,		CONFIG : 'N U T, 0, 0, 0',
	X =  23.370  mm,	Y =   -672.700  mm,	Z =   -248.196  mm,
	W =  90.000 deg,	P =   0.000 deg,	R =   90.000 deg
};
P[1189]{
   GP1:
	UF : 0, UT : 6,		CONFIG : 'N U T, 0, 0, 0',
	X =  23.847  mm,	Y =   -673.662  mm,	Z =   -248.005  mm,
	W =  90.000 deg,	P =   0.000 deg,	R =   90.000 deg
};
P[1190]{
   GP1:
	UF : 0, UT : 6,		CONFIG : 'N U T, 0, 0, 0',
	X =  25.377  mm,	Y =   -676.196  mm,	Z =   -248.169  mm,
	W =  90.000 deg,	P =   0.000 deg,	R =   90.000 deg
};
P[1191]{
   GP1:
	UF : 0, UT : 6,		CONFIG : 'N U T, 0, 0, 0',
	X =  25.859  mm,	Y =   -677.020  mm,	Z =   -248.181  mm,
	W =  90.000 deg,	P =   0.000 deg,	R =   90.000 deg
};
P[1192]{
   GP1:
	UF : 0, UT : 6,		CONFIG : 'N U T, 0, 0, 0',
	X =  27.557  mm,	Y =   -679.913  mm,	Z =   -248.248  mm,
	W =  90.000 deg,	P =   0.000 deg,	R =   90.000 deg
};
P[1193]{
   GP1:
	UF : 0, UT : 6,		CONFIG : 'N U T, 0, 0, 0',
	X =  27.859  mm,	Y =   -680.569  mm,	Z =   -248.060  mm,
	W =  90.000 deg,	P =   0.000 deg,	R =   90.000 deg
};
P[1194]{
   GP1:
	UF : 0, UT : 6,		CONFIG : 'N U T, 0, 0, 0',
	X =  29.538  mm,	Y =   -683.489  mm,	Z =   -248.044  mm,
	W =  90.000 deg,	P =   0.000 deg,	R =   90.000 deg
};
P[1195]{
   GP1:
	UF : 0, UT : 6,		CONFIG : 'N U T, 0, 0, 0',
	X =  30.041  mm,	Y =   -684.566  mm,	Z =   -247.758  mm,
	W =  90.000 deg,	P =   0.000 deg,	R =   90.000 deg
};
P[1196]{
   GP1:
	UF : 0, UT : 6,		CONFIG : 'N U T, 0, 0, 0',
	X =  32.655  mm,	Y =   -688.828  mm,	Z =   -248.129  mm,
	W =  90.000 deg,	P =   0.000 deg,	R =   90.000 deg
};
P[1197]{
   GP1:
	UF : 0, UT : 6,		CONFIG : 'N U T, 0, 0, 0',
	X =  32.992  mm,	Y =   -689.638  mm,	Z =   -247.812  mm,
	W =  90.000 deg,	P =   0.000 deg,	R =   90.000 deg
};
P[1198]{
   GP1:
	UF : 0, UT : 6,		CONFIG : 'N U T, 0, 0, 0',
	X =  33.516  mm,	Y =   -690.330  mm,	Z =   -248.114  mm,
	W =  90.000 deg,	P =   0.000 deg,	R =   90.000 deg
};
P[1199]{
   GP1:
	UF : 0, UT : 6,		CONFIG : 'N U T, 0, 0, 0',
	X =  35.670  mm,	Y =   -693.975  mm,	Z =   -248.235  mm,
	W =  90.000 deg,	P =   0.000 deg,	R =   90.000 deg
};
P[1200]{
   GP1:
	UF : 0, UT : 6,		CONFIG : 'N U T, 0, 0, 0',
	X =  37.981  mm,	Y =   -697.829  mm,	Z =   -247.791  mm,
	W =  90.000 deg,	P =   0.000 deg,	R =   90.000 deg
};
P[1201]{
   GP1:
	UF : 0, UT : 6,		CONFIG : 'N U T, 0, 0, 0',
	X =  40.056  mm,	Y =   -699.763  mm,	Z =   -248.051  mm,
	W =  90.000 deg,	P =   0.000 deg,	R =   90.000 deg
};
P[1202]{
   GP1:
	UF : 0, UT : 6,		CONFIG : 'N U T, 0, 0, 0',
	X =  41.424  mm,	Y =   -700.936  mm,	Z =   -247.777  mm,
	W =  90.000 deg,	P =   0.000 deg,	R =   90.000 deg
};
P[1203]{
   GP1:
	UF : 0, UT : 6,		CONFIG : 'N U T, 0, 0, 0',
	X =  43.211  mm,	Y =   -701.645  mm,	Z =   -248.228  mm,
	W =  90.000 deg,	P =   0.000 deg,	R =   90.000 deg
};
P[1204]{
   GP1:
	UF : 0, UT : 6,		CONFIG : 'N U T, 0, 0, 0',
	X =  46.506  mm,	Y =   -702.778  mm,	Z =   -247.853  mm,
	W =  90.000 deg,	P =   0.000 deg,	R =   90.000 deg
};
P[1205]{
   GP1:
	UF : 0, UT : 6,		CONFIG : 'N U T, 0, 0, 0',
	X =  49.902  mm,	Y =   -702.692  mm,	Z =   -248.175  mm,
	W =  90.000 deg,	P =   0.000 deg,	R =   90.000 deg
};
P[1206]{
   GP1:
	UF : 0, UT : 6,		CONFIG : 'N U T, 0, 0, 0',
	X =  52.498  mm,	Y =   -702.177  mm,	Z =   -248.089  mm,
	W =  90.000 deg,	P =   0.000 deg,	R =   90.000 deg
};
P[1207]{
   GP1:
	UF : 0, UT : 6,		CONFIG : 'N U T, 0, 0, 0',
	X =  53.598  mm,	Y =   -701.701  mm,	Z =   -248.206  mm,
	W =  90.000 deg,	P =   0.000 deg,	R =   90.000 deg
};
P[1208]{
   GP1:
	UF : 0, UT : 6,		CONFIG : 'N U T, 0, 0, 0',
	X =  57.828  mm,	Y =   -699.680  mm,	Z =   -247.792  mm,
	W =  90.000 deg,	P =   0.000 deg,	R =   90.000 deg
};
P[1209]{
   GP1:
	UF : 0, UT : 6,		CONFIG : 'N U T, 0, 0, 0',
	X =  59.459  mm,	Y =   -698.583  mm,	Z =   -248.167  mm,
	W =  90.000 deg,	P =   0.000 deg,	R =   90.000 deg
};
P[1210]{
   GP1:
	UF : 0, UT : 6,		CONFIG : 'N U T, 0, 0, 0',
	X =  60.293  mm,	Y =   -698.132  mm,	Z =   -248.095  mm,
	W =  90.000 deg,	P =   0.000 deg,	R =   90.000 deg
};
P[1211]{
   GP1:
	UF : 0, UT : 6,		CONFIG : 'N U T, 0, 0, 0',
	X =  63.529  mm,	Y =   -696.255  mm,	Z =   -248.116  mm,
	W =  90.000 deg,	P =   0.000 deg,	R =   90.000 deg
};
P[1212]{
   GP1:
	UF : 0, UT : 6,		CONFIG : 'N U T, 0, 0, 0',
	X =  67.009  mm,	Y =   -694.231  mm,	Z =   -248.150  mm,
	W =  90.000 deg,	P =   0.000 deg,	R =   90.000 deg
};
P[1213]{
   GP1:
	UF : 0, UT : 6,		CONFIG : 'N U T, 0, 0, 0',
	X =  68.551  mm,	Y =   -693.431  mm,	Z =   -247.933  mm,
	W =  90.000 deg,	P =   0.000 deg,	R =   90.000 deg
};
P[1214]{
   GP1:
	UF : 0, UT : 6,		CONFIG : 'N U T, 0, 0, 0',
	X =  69.566  mm,	Y =   -692.788  mm,	Z =   -248.069  mm,
	W =  90.000 deg,	P =   0.000 deg,	R =   90.000 deg
};
P[1215]{
   GP1:
	UF : 0, UT : 6,		CONFIG : 'N U T, 0, 0, 0',
	X =  70.714  mm,	Y =   -692.146  mm,	Z =   -248.019  mm,
	W =  90.000 deg,	P =   0.000 deg,	R =   90.000 deg
};
P[1216]{
   GP1:
	UF : 0, UT : 6,		CONFIG : 'N U T, 0, 0, 0',
	X =  71.313  mm,	Y =   -691.767  mm,	Z =   -248.098  mm,
	W =  90.000 deg,	P =   0.000 deg,	R =   90.000 deg
};
P[1217]{
   GP1:
	UF : 0, UT : 6,		CONFIG : 'N U T, 0, 0, 0',
	X =  72.438  mm,	Y =   -691.181  mm,	Z =   -247.946  mm,
	W =  90.000 deg,	P =   0.000 deg,	R =   90.000 deg
};
P[1218]{
   GP1:
	UF : 0, UT : 6,		CONFIG : 'N U T, 0, 0, 0',
	X =  75.268  mm,	Y =   -689.445  mm,	Z =   -248.191  mm,
	W =  90.000 deg,	P =   0.000 deg,	R =   90.000 deg
};
P[1219]{
   GP1:
	UF : 0, UT : 6,		CONFIG : 'N U T, 0, 0, 0',
	X =  76.260  mm,	Y =   -689.013  mm,	Z =   -247.850  mm,
	W =  90.000 deg,	P =   0.000 deg,	R =   90.000 deg
};
P[1220]{
   GP1:
	UF : 0, UT : 6,		CONFIG : 'N U T, 0, 0, 0',
	X =  81.444  mm,	Y =   -685.955  mm,	Z =   -248.010  mm,
	W =  90.000 deg,	P =   0.000 deg,	R =   90.000 deg
};
P[1221]{
   GP1:
	UF : 0, UT : 6,		CONFIG : 'N U T, 0, 0, 0',
	X =  82.162  mm,	Y =   -685.463  mm,	Z =   -248.197  mm,
	W =  90.000 deg,	P =   0.000 deg,	R =   90.000 deg
};
P[1222]{
   GP1:
	UF : 0, UT : 6,		CONFIG : 'N U T, 0, 0, 0',
	X =  83.825  mm,	Y =   -684.629  mm,	Z =   -247.891  mm,
	W =  90.000 deg,	P =   0.000 deg,	R =   90.000 deg
};
P[1223]{
   GP1:
	UF : 0, UT : 6,		CONFIG : 'N U T, 0, 0, 0',
	X =  88.339  mm,	Y =   -682.037  mm,	Z =   -247.856  mm,
	W =  90.000 deg,	P =   0.000 deg,	R =   90.000 deg
};
P[1224]{
   GP1:
	UF : 0, UT : 6,		CONFIG : 'N U T, 0, 0, 0',
	X =  90.188  mm,	Y =   -680.850  mm,	Z =   -248.145  mm,
	W =  90.000 deg,	P =   0.000 deg,	R =   90.000 deg
};
P[1225]{
   GP1:
	UF : 0, UT : 6,		CONFIG : 'N U T, 0, 0, 0',
	X =  91.201  mm,	Y =   -680.262  mm,	Z =   -248.151  mm,
	W =  90.000 deg,	P =   0.000 deg,	R =   90.000 deg
};
P[1226]{
   GP1:
	UF : 0, UT : 6,		CONFIG : 'N U T, 0, 0, 0',
	X =  92.454  mm,	Y =   -679.566  mm,	Z =   -248.086  mm,
	W =  90.000 deg,	P =   0.000 deg,	R =   90.000 deg
};
P[1227]{
   GP1:
	UF : 0, UT : 6,		CONFIG : 'N U T, 0, 0, 0',
	X =  95.464  mm,	Y =   -677.886  mm,	Z =   -247.945  mm,
	W =  90.000 deg,	P =   0.000 deg,	R =   90.000 deg
};
P[1228]{
   GP1:
	UF : 0, UT : 6,		CONFIG : 'N U T, 0, 0, 0',
	X =  99.928  mm,	Y =   -675.329  mm,	Z =   -247.897  mm,
	W =  90.000 deg,	P =   0.000 deg,	R =   90.000 deg
};
P[1229]{
   GP1:
	UF : 0, UT : 6,		CONFIG : 'N U T, 0, 0, 0',
	X =  102.048  mm,	Y =   -674.136  mm,	Z =   -247.820  mm,
	W =  90.000 deg,	P =   0.000 deg,	R =   90.000 deg
};
P[1230]{
   GP1:
	UF : 0, UT : 6,		CONFIG : 'N U T, 0, 0, 0',
	X =  106.132  mm,	Y =   -671.752  mm,	Z =   -247.882  mm,
	W =  90.000 deg,	P =   0.000 deg,	R =   90.000 deg
};
P[1231]{
   GP1:
	UF : 0, UT : 6,		CONFIG : 'N U T, 0, 0, 0',
	X =  106.812  mm,	Y =   -671.313  mm,	Z =   -247.996  mm,
	W =  90.000 deg,	P =   0.000 deg,	R =   90.000 deg
};
P[1232]{
   GP1:
	UF : 0, UT : 6,		CONFIG : 'N U T, 0, 0, 0',
	X =  108.511  mm,	Y =   -670.372  mm,	Z =   -247.899  mm,
	W =  90.000 deg,	P =   0.000 deg,	R =   90.000 deg
};
P[1233]{
   GP1:
	UF : 0, UT : 6,		CONFIG : 'N U T, 0, 0, 0',
	X =  110.558  mm,	Y =   -669.071  mm,	Z =   -248.188  mm,
	W =  90.000 deg,	P =   0.000 deg,	R =   90.000 deg
};
P[1234]{
   GP1:
	UF : 0, UT : 6,		CONFIG : 'N U T, 0, 0, 0',
	X =  111.510  mm,	Y =   -668.611  mm,	Z =   -247.969  mm,
	W =  90.000 deg,	P =   0.000 deg,	R =   90.000 deg
};
P[1235]{
   GP1:
	UF : 0, UT : 6,		CONFIG : 'N U T, 0, 0, 0',
	X =  112.767  mm,	Y =   -667.901  mm,	Z =   -247.933  mm,
	W =  90.000 deg,	P =   0.000 deg,	R =   90.000 deg
};
P[1236]{
   GP1:
	UF : 0, UT : 6,		CONFIG : 'N U T, 0, 0, 0',
	X =  114.098  mm,	Y =   -667.172  mm,	Z =   -247.835  mm,
	W =  90.000 deg,	P =   0.000 deg,	R =   90.000 deg
};
P[1237]{
   GP1:
	UF : 0, UT : 6,		CONFIG : 'N U T, 0, 0, 0',
	X =  115.371  mm,	Y =   -666.357  mm,	Z =   -248.029  mm,
	W =  90.000 deg,	P =   0.000 deg,	R =   90.000 deg
};
P[1238]{
   GP1:
	UF : 0, UT : 6,		CONFIG : 'N U T, 0, 0, 0',
	X =  116.918  mm,	Y =   -665.400  mm,	Z =   -248.184  mm,
	W =  90.000 deg,	P =   0.000 deg,	R =   90.000 deg
};
P[1239]{
   GP1:
	UF : 0, UT : 6,		CONFIG : 'N U T, 0, 0, 0',
	X =  117.618  mm,	Y =   -665.165  mm,	Z =   -247.773  mm,
	W =  90.000 deg,	P =   0.000 deg,	R =   90.000 deg
};
P[1240]{
   GP1:
	UF : 0, UT : 6,		CONFIG : 'N U T, 0, 0, 0',
	X =  118.761  mm,	Y =   -664.379  mm,	Z =   -248.080  mm,
	W =  90.000 deg,	P =   0.000 deg,	R =   90.000 deg
};
P[1241]{
   GP1:
	UF : 0, UT : 6,		CONFIG : 'N U T, 0, 0, 0',
	X =  119.542  mm,	Y =   -663.909  mm,	Z =   -248.128  mm,
	W =  90.000 deg,	P =   0.000 deg,	R =   90.000 deg
};
P[1242]{
   GP1:
	UF : 0, UT : 6,		CONFIG : 'N U T, 0, 0, 0',
	X =  120.346  mm,	Y =   -663.441  mm,	Z =   -248.136  mm,
	W =  90.000 deg,	P =   0.000 deg,	R =   90.000 deg
};
P[1243]{
   GP1:
	UF : 0, UT : 6,		CONFIG : 'N U T, 0, 0, 0',
	X =  121.285  mm,	Y =   -663.031  mm,	Z =   -247.815  mm,
	W =  90.000 deg,	P =   0.000 deg,	R =   90.000 deg
};
P[1244]{
   GP1:
	UF : 0, UT : 6,		CONFIG : 'N U T, 0, 0, 0',
	X =  121.809  mm,	Y =   -662.589  mm,	Z =   -248.153  mm,
	W =  90.000 deg,	P =   0.000 deg,	R =   90.000 deg
};
P[1245]{
   GP1:
	UF : 0, UT : 6,		CONFIG : 'N U T, 0, 0, 0',
	X =  124.128  mm,	Y =   -661.331  mm,	Z =   -247.956  mm,
	W =  90.000 deg,	P =   0.000 deg,	R =   90.000 deg
};
P[1246]{
   GP1:
	UF : 0, UT : 6,		CONFIG : 'N U T, 0, 0, 0',
	X =  124.868  mm,	Y =   -660.806  mm,	Z =   -248.192  mm,
	W =  90.000 deg,	P =   0.000 deg,	R =   90.000 deg
};
P[1247]{
   GP1:
	UF : 0, UT : 6,		CONFIG : 'N U T, 0, 0, 0',
	X =  127.204  mm,	Y =   -659.612  mm,	Z =   -247.818  mm,
	W =  90.000 deg,	P =   0.000 deg,	R =   90.000 deg
};
P[1248]{
   GP1:
	UF : 0, UT : 6,		CONFIG : 'N U T, 0, 0, 0',
	X =  130.550  mm,	Y =   -657.558  mm,	Z =   -248.114  mm,
	W =  90.000 deg,	P =   0.000 deg,	R =   90.000 deg
};
P[1249]{
   GP1:
	UF : 0, UT : 6,		CONFIG : 'N U T, 0, 0, 0',
	X =  133.248  mm,	Y =   -656.091  mm,	Z =   -247.894  mm,
	W =  90.000 deg,	P =   0.000 deg,	R =   90.000 deg
};
P[1250]{
   GP1:
	UF : 0, UT : 6,		CONFIG : 'N U T, 0, 0, 0',
	X =  133.901  mm,	Y =   -655.752  mm,	Z =   -247.802  mm,
	W =  90.000 deg,	P =   0.000 deg,	R =   90.000 deg
};
P[1251]{
   GP1:
	UF : 0, UT : 6,		CONFIG : 'N U T, 0, 0, 0',
	X =  136.252  mm,	Y =   -654.232  mm,	Z =   -248.194  mm,
	W =  90.000 deg,	P =   0.000 deg,	R =   90.000 deg
};
P[1252]{
   GP1:
	UF : 0, UT : 6,		CONFIG : 'N U T, 0, 0, 0',
	X =  138.038  mm,	Y =   -653.300  mm,	Z =   -247.956  mm,
	W =  90.000 deg,	P =   0.000 deg,	R =   90.000 deg
};
P[1253]{
   GP1:
	UF : 0, UT : 6,		CONFIG : 'N U T, 0, 0, 0',
	X =  139.134  mm,	Y =   -652.691  mm,	Z =   -247.897  mm,
	W =  90.000 deg,	P =   0.000 deg,	R =   90.000 deg
};
P[1254]{
   GP1:
	UF : 0, UT : 6,		CONFIG : 'N U T, 0, 0, 0',
	X =  139.855  mm,	Y =   -652.194  mm,	Z =   -248.094  mm,
	W =  90.000 deg,	P =   0.000 deg,	R =   90.000 deg
};
P[1255]{
   GP1:
	UF : 0, UT : 6,		CONFIG : 'N U T, 0, 0, 0',
	X =  143.057  mm,	Y =   -650.323  mm,	Z =   -248.145  mm,
	W =  90.000 deg,	P =   0.000 deg,	R =   90.000 deg
};
P[1256]{
   GP1:
	UF : 0, UT : 6,		CONFIG : 'N U T, 0, 0, 0',
	X =  144.000  mm,	Y =   -649.787  mm,	Z =   -248.127  mm,
	W =  90.000 deg,	P =   0.000 deg,	R =   90.000 deg
};
P[1257]{
   GP1:
	UF : 0, UT : 6,		CONFIG : 'N U T, 0, 0, 0',
	X =  145.130  mm,	Y =   -649.126  mm,	Z =   -248.147  mm,
	W =  90.000 deg,	P =   0.000 deg,	R =   90.000 deg
};
P[1258]{
   GP1:
	UF : 0, UT : 6,		CONFIG : 'N U T, 0, 0, 0',
	X =  146.095  mm,	Y =   -648.605  mm,	Z =   -248.061  mm,
	W =  90.000 deg,	P =   0.000 deg,	R =   90.000 deg
};
P[1259]{
   GP1:
	UF : 0, UT : 6,		CONFIG : 'N U T, 0, 0, 0',
	X =  147.553  mm,	Y =   -647.767  mm,	Z =   -248.052  mm,
	W =  90.000 deg,	P =   0.000 deg,	R =   90.000 deg
};
P[1260]{
   GP1:
	UF : 0, UT : 6,		CONFIG : 'N U T, 0, 0, 0',
	X =  148.698  mm,	Y =   -647.175  mm,	Z =   -247.883  mm,
	W =  90.000 deg,	P =   0.000 deg,	R =   90.000 deg
};
P[1261]{
   GP1:
	UF : 0, UT : 6,		CONFIG : 'N U T, 0, 0, 0',
	X =  149.961  mm,	Y =   -646.307  mm,	Z =   -248.219  mm,
	W =  90.000 deg,	P =   0.000 deg,	R =   90.000 deg
};
P[1262]{
   GP1:
	UF : 0, UT : 6,		CONFIG : 'N U T, 0, 0, 0',
	X =  150.911  mm,	Y =   -645.870  mm,	Z =   -247.949  mm,
	W =  90.000 deg,	P =   0.000 deg,	R =   90.000 deg
};
P[1263]{
   GP1:
	UF : 0, UT : 6,		CONFIG : 'N U T, 0, 0, 0',
	X =  151.621  mm,	Y =   -645.473  mm,	Z =   -247.918  mm,
	W =  90.000 deg,	P =   0.000 deg,	R =   90.000 deg
};
P[1264]{
   GP1:
	UF : 0, UT : 6,		CONFIG : 'N U T, 0, 0, 0',
	X =  152.843  mm,	Y =   -644.667  mm,	Z =   -248.162  mm,
	W =  90.000 deg,	P =   0.000 deg,	R =   90.000 deg
};
P[1265]{
   GP1:
	UF : 0, UT : 6,		CONFIG : 'N U T, 0, 0, 0',
	X =  155.926  mm,	Y =   -642.985  mm,	Z =   -247.924  mm,
	W =  90.000 deg,	P =   0.000 deg,	R =   90.000 deg
};
P[1266]{
   GP1:
	UF : 0, UT : 6,		CONFIG : 'N U T, 0, 0, 0',
	X =  157.162  mm,	Y =   -642.309  mm,	Z =   -247.829  mm,
	W =  90.000 deg,	P =   0.000 deg,	R =   90.000 deg
};
P[1267]{
   GP1:
	UF : 0, UT : 6,		CONFIG : 'N U T, 0, 0, 0',
	X =  158.193  mm,	Y =   -641.628  mm,	Z =   -248.038  mm,
	W =  90.000 deg,	P =   0.000 deg,	R =   90.000 deg
};
P[1268]{
   GP1:
	UF : 0, UT : 6,		CONFIG : 'N U T, 0, 0, 0',
	X =  162.791  mm,	Y =   -639.011  mm,	Z =   -247.948  mm,
	W =  90.000 deg,	P =   0.000 deg,	R =   90.000 deg
};
P[1269]{
   GP1:
	UF : 0, UT : 6,		CONFIG : 'N U T, 0, 0, 0',
	X =  163.366  mm,	Y =   -638.629  mm,	Z =   -248.070  mm,
	W =  90.000 deg,	P =   0.000 deg,	R =   90.000 deg
};
P[1270]{
   GP1:
	UF : 0, UT : 6,		CONFIG : 'N U T, 0, 0, 0',
	X =  164.338  mm,	Y =   -638.057  mm,	Z =   -248.096  mm,
	W =  90.000 deg,	P =   0.000 deg,	R =   90.000 deg
};
P[1271]{
   GP1:
	UF : 0, UT : 6,		CONFIG : 'N U T, 0, 0, 0',
	X =  166.149  mm,	Y =   -637.013  mm,	Z =   -248.091  mm,
	W =  90.000 deg,	P =   0.000 deg,	R =   90.000 deg
};
P[1272]{
   GP1:
	UF : 0, UT : 6,		CONFIG : 'N U T, 0, 0, 0',
	X =  166.768  mm,	Y =   -636.609  mm,	Z =   -248.204  mm,
	W =  90.000 deg,	P =   0.000 deg,	R =   90.000 deg
};
P[1273]{
   GP1:
	UF : 0, UT : 6,		CONFIG : 'N U T, 0, 0, 0',
	X =  170.822  mm,	Y =   -634.411  mm,	Z =   -247.859  mm,
	W =  90.000 deg,	P =   0.000 deg,	R =   90.000 deg
};
P[1274]{
   GP1:
	UF : 0, UT : 6,		CONFIG : 'N U T, 0, 0, 0',
	X =  172.271  mm,	Y =   -633.521  mm,	Z =   -247.986  mm,
	W =  90.000 deg,	P =   0.000 deg,	R =   90.000 deg
};
P[1275]{
   GP1:
	UF : 0, UT : 6,		CONFIG : 'N U T, 0, 0, 0',
	X =  173.229  mm,	Y =   -632.942  mm,	Z =   -248.050  mm,
	W =  90.000 deg,	P =   0.000 deg,	R =   90.000 deg
};
P[1276]{
   GP1:
	UF : 0, UT : 6,		CONFIG : 'N U T, 0, 0, 0',
	X =  173.874  mm,	Y =   -632.618  mm,	Z =   -247.933  mm,
	W =  90.000 deg,	P =   0.000 deg,	R =   90.000 deg
};
P[1277]{
   GP1:
	UF : 0, UT : 6,		CONFIG : 'N U T, 0, 0, 0',
	X =  174.774  mm,	Y =   -632.117  mm,	Z =   -247.889  mm,
	W =  90.000 deg,	P =   0.000 deg,	R =   90.000 deg
};
P[1278]{
   GP1:
	UF : 0, UT : 6,		CONFIG : 'N U T, 0, 0, 0',
	X =  175.268  mm,	Y =   -631.683  mm,	Z =   -248.246  mm,
	W =  90.000 deg,	P =   0.000 deg,	R =   90.000 deg
};
P[1279]{
   GP1:
	UF : 0, UT : 6,		CONFIG : 'N U T, 0, 0, 0',
	X =  176.225  mm,	Y =   -631.221  mm,	Z =   -248.027  mm,
	W =  90.000 deg,	P =   0.000 deg,	R =   90.000 deg
};
P[1280]{
   GP1:
	UF : 0, UT : 6,		CONFIG : 'N U T, 0, 0, 0',
	X =  180.531  mm,	Y =   -628.751  mm,	Z =   -247.988  mm,
	W =  90.000 deg,	P =   0.000 deg,	R =   90.000 deg
};
P[1281]{
   GP1:
	UF : 0, UT : 6,		CONFIG : 'N U T, 0, 0, 0',
	X =  182.115  mm,	Y =   -627.763  mm,	Z =   -248.168  mm,
	W =  90.000 deg,	P =   0.000 deg,	R =   90.000 deg
};
P[1282]{
   GP1:
	UF : 0, UT : 6,		CONFIG : 'N U T, 0, 0, 0',
	X =  183.204  mm,	Y =   -627.147  mm,	Z =   -248.137  mm,
	W =  90.000 deg,	P =   0.000 deg,	R =   90.000 deg
};
P[1283]{
   GP1:
	UF : 0, UT : 6,		CONFIG : 'N U T, 0, 0, 0',
	X =  183.925  mm,	Y =   -626.756  mm,	Z =   -248.073  mm,
	W =  90.000 deg,	P =   0.000 deg,	R =   90.000 deg
};
P[1284]{
   GP1:
	UF : 0, UT : 6,		CONFIG : 'N U T, 0, 0, 0',
	X =  185.279  mm,	Y =   -625.929  mm,	Z =   -248.185  mm,
	W =  90.000 deg,	P =   0.000 deg,	R =   90.000 deg
};
P[1285]{
   GP1:
	UF : 0, UT : 6,		CONFIG : 'N U T, 0, 0, 0',
	X =  186.525  mm,	Y =   -625.229  mm,	Z =   -248.139  mm,
	W =  90.000 deg,	P =   0.000 deg,	R =   90.000 deg
};
P[1286]{
   GP1:
	UF : 0, UT : 6,		CONFIG : 'N U T, 0, 0, 0',
	X =  189.282  mm,	Y =   -623.613  mm,	Z =   -248.195  mm,
	W =  90.000 deg,	P =   0.000 deg,	R =   90.000 deg
};
P[1287]{
   GP1:
	UF : 0, UT : 6,		CONFIG : 'N U T, 0, 0, 0',
	X =  195.128  mm,	Y =   -620.296  mm,	Z =   -248.054  mm,
	W =  90.000 deg,	P =   0.000 deg,	R =   90.000 deg
};
P[1288]{
   GP1:
	UF : 0, UT : 6,		CONFIG : 'N U T, 0, 0, 0',
	X =  196.317  mm,	Y =   -619.610  mm,	Z =   -248.052  mm,
	W =  90.000 deg,	P =   0.000 deg,	R =   90.000 deg
};
P[1289]{
   GP1:
	UF : 0, UT : 6,		CONFIG : 'N U T, 0, 0, 0',
	X =  199.877  mm,	Y =   -617.671  mm,	Z =   -247.770  mm,
	W =  90.000 deg,	P =   0.000 deg,	R =   90.000 deg
};
P[1290]{
   GP1:
	UF : 0, UT : 6,		CONFIG : 'N U T, 0, 0, 0',
	X =  200.882  mm,	Y =   -616.951  mm,	Z =   -248.110  mm,
	W =  90.000 deg,	P =   0.000 deg,	R =   90.000 deg
};
P[1291]{
   GP1:
	UF : 0, UT : 6,		CONFIG : 'N U T, 0, 0, 0',
	X =  202.702  mm,	Y =   -616.037  mm,	Z =   -247.776  mm,
	W =  90.000 deg,	P =   0.000 deg,	R =   90.000 deg
};
P[1292]{
   GP1:
	UF : 0, UT : 6,		CONFIG : 'N U T, 0, 0, 0',
	X =  204.218  mm,	Y =   -615.118  mm,	Z =   -247.884  mm,
	W =  90.000 deg,	P =   0.000 deg,	R =   90.000 deg
};
P[1293]{
   GP1:
	UF : 0, UT : 6,		CONFIG : 'N U T, 0, 0, 0',
	X =  205.265  mm,	Y =   -614.374  mm,	Z =   -248.222  mm,
	W =  90.000 deg,	P =   0.000 deg,	R =   90.000 deg
};
P[1294]{
   GP1:
	UF : 0, UT : 6,		CONFIG : 'N U T, 0, 0, 0',
	X =  209.280  mm,	Y =   -612.065  mm,	Z =   -248.199  mm,
	W =  90.000 deg,	P =   0.000 deg,	R =   90.000 deg
};
P[1295]{
   GP1:
	UF : 0, UT : 6,		CONFIG : 'N U T, 0, 0, 0',
	X =  210.238  mm,	Y =   -611.576  mm,	Z =   -248.045  mm,
	W =  90.000 deg,	P =   0.000 deg,	R =   90.000 deg
};
P[1296]{
   GP1:
	UF : 0, UT : 6,		CONFIG : 'N U T, 0, 0, 0',
	X =  211.137  mm,	Y =   -611.124  mm,	Z =   -247.881  mm,
	W =  90.000 deg,	P =   0.000 deg,	R =   90.000 deg
};
P[1297]{
   GP1:
	UF : 0, UT : 6,		CONFIG : 'N U T, 0, 0, 0',
	X =  212.061  mm,	Y =   -610.490  mm,	Z =   -248.124  mm,
	W =  90.000 deg,	P =   0.000 deg,	R =   90.000 deg
};
P[1298]{
   GP1:
	UF : 0, UT : 6,		CONFIG : 'N U T, 0, 0, 0',
	X =  214.997  mm,	Y =   -608.911  mm,	Z =   -247.843  mm,
	W =  90.000 deg,	P =   0.000 deg,	R =   90.000 deg
};
P[1299]{
   GP1:
	UF : 0, UT : 6,		CONFIG : 'N U T, 0, 0, 0',
	X =  215.840  mm,	Y =   -608.348  mm,	Z =   -248.028  mm,
	W =  90.000 deg,	P =   0.000 deg,	R =   90.000 deg
};
P[1300]{
   GP1:
	UF : 0, UT : 6,		CONFIG : 'N U T, 0, 0, 0',
	X =  217.212  mm,	Y =   -607.527  mm,	Z =   -248.098  mm,
	W =  90.000 deg,	P =   0.000 deg,	R =   90.000 deg
};
P[1301]{
   GP1:
	UF : 0, UT : 6,		CONFIG : 'N U T, 0, 0, 0',
	X =  218.505  mm,	Y =   -606.758  mm,	Z =   -248.150  mm,
	W =  90.000 deg,	P =   0.000 deg,	R =   90.000 deg
};
P[1302]{
   GP1:
	UF : 0, UT : 6,		CONFIG : 'N U T, 0, 0, 0',
	X =  219.370  mm,	Y =   -606.373  mm,	Z =   -247.873  mm,
	W =  90.000 deg,	P =   0.000 deg,	R =   90.000 deg
};
P[1303]{
   GP1:
	UF : 0, UT : 6,		CONFIG : 'N U T, 0, 0, 0',
	X =  221.697  mm,	Y =   -604.929  mm,	Z =   -248.119  mm,
	W =  90.000 deg,	P =   0.000 deg,	R =   90.000 deg
};
P[1304]{
   GP1:
	UF : 0, UT : 6,		CONFIG : 'N U T, 0, 0, 0',
	X =  223.052  mm,	Y =   -604.196  mm,	Z =   -248.000  mm,
	W =  90.000 deg,	P =   0.000 deg,	R =   90.000 deg
};
P[1305]{
   GP1:
	UF : 0, UT : 6,		CONFIG : 'N U T, 0, 0, 0',
	X =  224.713  mm,	Y =   -603.137  mm,	Z =   -248.242  mm,
	W =  90.000 deg,	P =   0.000 deg,	R =   90.000 deg
};
P[1306]{
   GP1:
	UF : 0, UT : 6,		CONFIG : 'N U T, 0, 0, 0',
	X =  226.437  mm,	Y =   -602.204  mm,	Z =   -248.090  mm,
	W =  90.000 deg,	P =   0.000 deg,	R =   90.000 deg
};
P[1307]{
   GP1:
	UF : 0, UT : 6,		CONFIG : 'N U T, 0, 0, 0',
	X =  227.299  mm,	Y =   -601.670  mm,	Z =   -248.178  mm,
	W =  90.000 deg,	P =   0.000 deg,	R =   90.000 deg
};
P[1308]{
   GP1:
	UF : 0, UT : 6,		CONFIG : 'N U T, 0, 0, 0',
	X =  228.163  mm,	Y =   -601.174  mm,	Z =   -248.170  mm,
	W =  90.000 deg,	P =   0.000 deg,	R =   90.000 deg
};
P[1309]{
   GP1:
	UF : 0, UT : 6,		CONFIG : 'N U T, 0, 0, 0',
	X =  228.807  mm,	Y =   -600.934  mm,	Z =   -247.850  mm,
	W =  90.000 deg,	P =   0.000 deg,	R =   90.000 deg
};
P[1310]{
   GP1:
	UF : 0, UT : 6,		CONFIG : 'N U T, 0, 0, 0',
	X =  231.504  mm,	Y =   -599.317  mm,	Z =   -247.996  mm,
	W =  90.000 deg,	P =   0.000 deg,	R =   90.000 deg
};
P[1311]{
   GP1:
	UF : 0, UT : 6,		CONFIG : 'N U T, 0, 0, 0',
	X =  232.965  mm,	Y =   -598.376  mm,	Z =   -248.232  mm,
	W =  90.000 deg,	P =   0.000 deg,	R =   90.000 deg
};
P[1312]{
   GP1:
	UF : 0, UT : 6,		CONFIG : 'N U T, 0, 0, 0',
	X =  233.950  mm,	Y =   -597.854  mm,	Z =   -248.118  mm,
	W =  90.000 deg,	P =   0.000 deg,	R =   90.000 deg
};
P[1313]{
   GP1:
	UF : 0, UT : 6,		CONFIG : 'N U T, 0, 0, 0',
	X =  235.645  mm,	Y =   -596.825  mm,	Z =   -248.241  mm,
	W =  90.000 deg,	P =   0.000 deg,	R =   90.000 deg
};
P[1314]{
   GP1:
	UF : 0, UT : 6,		CONFIG : 'N U T, 0, 0, 0',
	X =  236.759  mm,	Y =   -596.265  mm,	Z =   -248.039  mm,
	W =  90.000 deg,	P =   0.000 deg,	R =   90.000 deg
};
P[1315]{
   GP1:
	UF : 0, UT : 6,		CONFIG : 'N U T, 0, 0, 0',
	X =  238.258  mm,	Y =   -595.340  mm,	Z =   -248.183  mm,
	W =  90.000 deg,	P =   0.000 deg,	R =   90.000 deg
};
P[1316]{
   GP1:
	UF : 0, UT : 6,		CONFIG : 'N U T, 0, 0, 0',
	X =  239.102  mm,	Y =   -594.830  mm,	Z =   -248.239  mm,
	W =  90.000 deg,	P =   0.000 deg,	R =   90.000 deg
};
P[1317]{
   GP1:
	UF : 0, UT : 6,		CONFIG : 'N U T, 0, 0, 0',
	X =  240.792  mm,	Y =   -593.995  mm,	Z =   -247.898  mm,
	W =  90.000 deg,	P =   0.000 deg,	R =   90.000 deg
};
P[1318]{
   GP1:
	UF : 0, UT : 6,		CONFIG : 'N U T, 0, 0, 0',
	X =  242.450  mm,	Y =   -592.901  mm,	Z =   -248.228  mm,
	W =  90.000 deg,	P =   0.000 deg,	R =   90.000 deg
};
P[1319]{
   GP1:
	UF : 0, UT : 6,		CONFIG : 'N U T, 0, 0, 0',
	X =  243.435  mm,	Y =   -592.498  mm,	Z =   -247.826  mm,
	W =  90.000 deg,	P =   0.000 deg,	R =   90.000 deg
};
P[1320]{
   GP1:
	UF : 0, UT : 6,		CONFIG : 'N U T, 0, 0, 0',
	X =  245.817  mm,	Y =   -590.948  mm,	Z =   -248.250  mm,
	W =  90.000 deg,	P =   0.000 deg,	R =   90.000 deg
};
P[1321]{
   GP1:
	UF : 0, UT : 6,		CONFIG : 'N U T, 0, 0, 0',
	X =  246.775  mm,	Y =   -590.418  mm,	Z =   -248.195  mm,
	W =  90.000 deg,	P =   0.000 deg,	R =   90.000 deg
};
P[1322]{
   GP1:
	UF : 0, UT : 6,		CONFIG : 'N U T, 0, 0, 0',
	X =  249.172  mm,	Y =   -589.049  mm,	Z =   -248.158  mm,
	W =  90.000 deg,	P =   0.000 deg,	R =   90.000 deg
};
P[1323]{
   GP1:
	UF : 0, UT : 6,		CONFIG : 'N U T, 0, 0, 0',
	X =  252.750  mm,	Y =   -586.953  mm,	Z =   -248.231  mm,
	W =  90.000 deg,	P =   0.000 deg,	R =   90.000 deg
};
P[1324]{
   GP1:
	UF : 0, UT : 6,		CONFIG : 'N U T, 0, 0, 0',
	X =  254.249  mm,	Y =   -586.123  mm,	Z =   -248.143  mm,
	W =  90.000 deg,	P =   0.000 deg,	R =   90.000 deg
};
P[1325]{
   GP1:
	UF : 0, UT : 6,		CONFIG : 'N U T, 0, 0, 0',
	X =  255.166  mm,	Y =   -585.568  mm,	Z =   -248.207  mm,
	W =  90.000 deg,	P =   0.000 deg,	R =   90.000 deg
};
P[1326]{
   GP1:
	UF : 0, UT : 6,		CONFIG : 'N U T, 0, 0, 0',
	X =  257.700  mm,	Y =   -584.133  mm,	Z =   -248.138  mm,
	W =  90.000 deg,	P =   0.000 deg,	R =   90.000 deg
};
P[1327]{
   GP1:
	UF : 0, UT : 6,		CONFIG : 'N U T, 0, 0, 0',
	X =  260.577  mm,	Y =   -582.561  mm,	Z =   -247.922  mm,
	W =  90.000 deg,	P =   0.000 deg,	R =   90.000 deg
};
P[1328]{
   GP1:
	UF : 0, UT : 6,		CONFIG : 'N U T, 0, 0, 0',
	X =  262.655  mm,	Y =   -581.326  mm,	Z =   -248.006  mm,
	W =  90.000 deg,	P =   0.000 deg,	R =   90.000 deg
};
P[1329]{
   GP1:
	UF : 0, UT : 6,		CONFIG : 'N U T, 0, 0, 0',
	X =  263.466  mm,	Y =   -580.857  mm,	Z =   -248.009  mm,
	W =  90.000 deg,	P =   0.000 deg,	R =   90.000 deg
};
P[1330]{
   GP1:
	UF : 0, UT : 6,		CONFIG : 'N U T, 0, 0, 0',
	X =  264.279  mm,	Y =   -580.326  mm,	Z =   -248.156  mm,
	W =  90.000 deg,	P =   0.000 deg,	R =   90.000 deg
};
P[1331]{
   GP1:
	UF : 0, UT : 6,		CONFIG : 'N U T, 0, 0, 0',
	X =  264.924  mm,	Y =   -580.010  mm,	Z =   -248.023  mm,
	W =  90.000 deg,	P =   0.000 deg,	R =   90.000 deg
};
P[1332]{
   GP1:
	UF : 0, UT : 6,		CONFIG : 'N U T, 0, 0, 0',
	X =  266.431  mm,	Y =   -579.203  mm,	Z =   -247.870  mm,
	W =  90.000 deg,	P =   0.000 deg,	R =   90.000 deg
};
P[1333]{
   GP1:
	UF : 0, UT : 6,		CONFIG : 'N U T, 0, 0, 0',
	X =  267.122  mm,	Y =   -578.691  mm,	Z =   -248.144  mm,
	W =  90.000 deg,	P =   0.000 deg,	R =   90.000 deg
};
P[1334]{
   GP1:
	UF : 0, UT : 6,		CONFIG : 'N U T, 0, 0, 0',
	X =  269.994  mm,	Y =   -577.182  mm,	Z =   -247.782  mm,
	W =  90.000 deg,	P =   0.000 deg,	R =   90.000 deg
};
P[1335]{
   GP1:
	UF : 0, UT : 6,		CONFIG : 'N U T, 0, 0, 0',
	X =  271.954  mm,	Y =   -575.895  mm,	Z =   -248.156  mm,
	W =  90.000 deg,	P =   0.000 deg,	R =   90.000 deg
};
P[1336]{
   GP1:
	UF : 0, UT : 6,		CONFIG : 'N U T, 0, 0, 0',
	X =  273.333  mm,	Y =   -575.233  mm,	Z =   -247.829  mm,
	W =  90.000 deg,	P =   0.000 deg,	R =   90.000 deg
};
P[1337]{
   GP1:
	UF : 0, UT : 6,		CONFIG : 'N U T, 0, 0, 0',
	X =  274.468  mm,	Y =   -574.438  mm,	Z =   -248.171  mm,
	W =  90.000 deg,	P =   0.000 deg,	R =   90.000 deg
};
P[1338]{
   GP1:
	UF : 0, UT : 6,		CONFIG : 'N U T, 0, 0, 0',
	X =  277.572  mm,	Y =   -572.786  mm,	Z =   -247.831  mm,
	W =  90.000 deg,	P =   0.000 deg,	R =   90.000 deg
};
P[1339]{
   GP1:
	UF : 0, UT : 6,		CONFIG : 'N U T, 0, 0, 0',
	X =  278.731  mm,	Y =   -572.117  mm,	Z =   -247.827  mm,
	W =  90.000 deg,	P =   0.000 deg,	R =   90.000 deg
};
P[1340]{
   GP1:
	UF : 0, UT : 6,		CONFIG : 'N U T, 0, 0, 0',
	X =  280.262  mm,	Y =   -571.226  mm,	Z =   -247.847  mm,
	W =  90.000 deg,	P =   0.000 deg,	R =   90.000 deg
};
P[1341]{
   GP1:
	UF : 0, UT : 6,		CONFIG : 'N U T, 0, 0, 0',
	X =  283.626  mm,	Y =   -569.221  mm,	Z =   -247.997  mm,
	W =  90.000 deg,	P =   0.000 deg,	R =   90.000 deg
};
P[1342]{
   GP1:
	UF : 0, UT : 6,		CONFIG : 'N U T, 0, 0, 0',
	X =  284.454  mm,	Y =   -568.792  mm,	Z =   -247.879  mm,
	W =  90.000 deg,	P =   0.000 deg,	R =   90.000 deg
};
P[1343]{
   GP1:
	UF : 0, UT : 6,		CONFIG : 'N U T, 0, 0, 0',
	X =  285.895  mm,	Y =   -567.870  mm,	Z =   -248.098  mm,
	W =  90.000 deg,	P =   0.000 deg,	R =   90.000 deg
};
P[1344]{
   GP1:
	UF : 0, UT : 6,		CONFIG : 'N U T, 0, 0, 0',
	X =  287.003  mm,	Y =   -567.189  mm,	Z =   -248.198  mm,
	W =  90.000 deg,	P =   0.000 deg,	R =   90.000 deg
};
P[1345]{
   GP1:
	UF : 0, UT : 6,		CONFIG : 'N U T, 0, 0, 0',
	X =  288.110  mm,	Y =   -566.532  mm,	Z =   -248.241  mm,
	W =  90.000 deg,	P =   0.000 deg,	R =   90.000 deg
};
P[1346]{
   GP1:
	UF : 0, UT : 6,		CONFIG : 'N U T, 0, 0, 0',
	X =  290.009  mm,	Y =   -565.496  mm,	Z =   -248.093  mm,
	W =  90.000 deg,	P =   0.000 deg,	R =   90.000 deg
};
P[1347]{
   GP1:
	UF : 0, UT : 6,		CONFIG : 'N U T, 0, 0, 0',
	X =  292.721  mm,	Y =   -564.015  mm,	Z =   -247.889  mm,
	W =  90.000 deg,	P =   0.000 deg,	R =   90.000 deg
};
P[1348]{
   GP1:
	UF : 0, UT : 6,		CONFIG : 'N U T, 0, 0, 0',
	X =  296.720  mm,	Y =   -561.736  mm,	Z =   -247.814  mm,
	W =  90.000 deg,	P =   0.000 deg,	R =   90.000 deg
};
P[1349]{
   GP1:
	UF : 0, UT : 6,		CONFIG : 'N U T, 0, 0, 0',
	X =  297.712  mm,	Y =   -561.068  mm,	Z =   -248.048  mm,
	W =  90.000 deg,	P =   0.000 deg,	R =   90.000 deg
};
P[1350]{
   GP1:
	UF : 0, UT : 6,		CONFIG : 'N U T, 0, 0, 0',
	X =  300.447  mm,	Y =   -559.465  mm,	Z =   -248.105  mm,
	W =  90.000 deg,	P =   0.000 deg,	R =   90.000 deg
};
P[1351]{
   GP1:
	UF : 0, UT : 6,		CONFIG : 'N U T, 0, 0, 0',
	X =  301.670  mm,	Y =   -558.819  mm,	Z =   -247.960  mm,
	W =  90.000 deg,	P =   0.000 deg,	R =   90.000 deg
};
P[1352]{
   GP1:
	UF : 0, UT : 6,		CONFIG : 'N U T, 0, 0, 0',
	X =  303.943  mm,	Y =   -557.486  mm,	Z =   -248.008  mm,
	W =  90.000 deg,	P =   0.000 deg,	R =   90.000 deg
};
P[1353]{
   GP1:
	UF : 0, UT : 6,		CONFIG : 'N U T, 0, 0, 0',
	X =  305.058  mm,	Y =   -556.901  mm,	Z =   -247.867  mm,
	W =  90.000 deg,	P =   0.000 deg,	R =   90.000 deg
};
P[1354]{
   GP1:
	UF : 0, UT : 6,		CONFIG : 'N U T, 0, 0, 0',
	X =  305.967  mm,	Y =   -556.219  mm,	Z =   -248.248  mm,
	W =  90.000 deg,	P =   0.000 deg,	R =   90.000 deg
};
P[1355]{
   GP1:
	UF : 0, UT : 6,		CONFIG : 'N U T, 0, 0, 0',
	X =  310.714  mm,	Y =   -553.489  mm,	Z =   -248.221  mm,
	W =  90.000 deg,	P =   0.000 deg,	R =   90.000 deg
};
P[1356]{
   GP1:
	UF : 0, UT : 6,		CONFIG : 'N U T, 0, 0, 0',
	X =  311.888  mm,	Y =   -552.938  mm,	Z =   -247.914  mm,
	W =  90.000 deg,	P =   0.000 deg,	R =   90.000 deg
};
P[1357]{
   GP1:
	UF : 0, UT : 6,		CONFIG : 'N U T, 0, 0, 0',
	X =  312.963  mm,	Y =   -552.289  mm,	Z =   -247.982  mm,
	W =  90.000 deg,	P =   0.000 deg,	R =   90.000 deg
};
P[1358]{
   GP1:
	UF : 0, UT : 6,		CONFIG : 'N U T, 0, 0, 0',
	X =  315.463  mm,	Y =   -550.763  mm,	Z =   -248.181  mm,
	W =  90.000 deg,	P =   0.000 deg,	R =   90.000 deg
};
P[1359]{
   GP1:
	UF : 0, UT : 6,		CONFIG : 'N U T, 0, 0, 0',
	X =  317.740  mm,	Y =   -549.454  mm,	Z =   -248.168  mm,
	W =  90.000 deg,	P =   0.000 deg,	R =   90.000 deg
};
P[1360]{
   GP1:
	UF : 0, UT : 6,		CONFIG : 'N U T, 0, 0, 0',
	X =  318.973  mm,	Y =   -548.775  mm,	Z =   -248.090  mm,
	W =  90.000 deg,	P =   0.000 deg,	R =   90.000 deg
};
P[1361]{
   GP1:
	UF : 0, UT : 6,		CONFIG : 'N U T, 0, 0, 0',
	X =  319.887  mm,	Y =   -548.258  mm,	Z =   -248.061  mm,
	W =  90.000 deg,	P =   0.000 deg,	R =   90.000 deg
};
P[1362]{
   GP1:
	UF : 0, UT : 6,		CONFIG : 'N U T, 0, 0, 0',
	X =  322.236  mm,	Y =   -546.963  mm,	Z =   -247.914  mm,
	W =  90.000 deg,	P =   0.000 deg,	R =   90.000 deg
};
P[1363]{
   GP1:
	UF : 0, UT : 6,		CONFIG : 'N U T, 0, 0, 0',
	X =  324.992  mm,	Y =   -545.303  mm,	Z =   -248.080  mm,
	W =  90.000 deg,	P =   0.000 deg,	R =   90.000 deg
};
P[1364]{
   GP1:
	UF : 0, UT : 6,		CONFIG : 'N U T, 0, 0, 0',
	X =  326.052  mm,	Y =   -544.823  mm,	Z =   -247.758  mm,
	W =  90.000 deg,	P =   0.000 deg,	R =   90.000 deg
};
P[1365]{
   GP1:
	UF : 0, UT : 6,		CONFIG : 'N U T, 0, 0, 0',
	X =  330.105  mm,	Y =   -542.391  mm,	Z =   -247.980  mm,
	W =  90.000 deg,	P =   0.000 deg,	R =   90.000 deg
};
P[1366]{
   GP1:
	UF : 0, UT : 6,		CONFIG : 'N U T, 0, 0, 0',
	X =  332.854  mm,	Y =   -540.693  mm,	Z =   -248.251  mm,
	W =  90.000 deg,	P =   0.000 deg,	R =   90.000 deg
};
P[1367]{
   GP1:
	UF : 0, UT : 6,		CONFIG : 'N U T, 0, 0, 0',
	X =  335.548  mm,	Y =   -539.269  mm,	Z =   -247.932  mm,
	W =  90.000 deg,	P =   0.000 deg,	R =   90.000 deg
};
P[1368]{
   GP1:
	UF : 0, UT : 6,		CONFIG : 'N U T, 0, 0, 0',
	X =  336.403  mm,	Y =   -538.703  mm,	Z =   -248.108  mm,
	W =  90.000 deg,	P =   0.000 deg,	R =   90.000 deg
};
P[1369]{
   GP1:
	UF : 0, UT : 6,		CONFIG : 'N U T, 0, 0, 0',
	X =  337.290  mm,	Y =   -538.144  mm,	Z =   -248.221  mm,
	W =  90.000 deg,	P =   0.000 deg,	R =   90.000 deg
};
P[1370]{
   GP1:
	UF : 0, UT : 6,		CONFIG : 'N U T, 0, 0, 0',
	X =  339.617  mm,	Y =   -536.867  mm,	Z =   -248.061  mm,
	W =  90.000 deg,	P =   0.000 deg,	R =   90.000 deg
};
P[1371]{
   GP1:
	UF : 0, UT : 6,		CONFIG : 'N U T, 0, 0, 0',
	X =  340.749  mm,	Y =   -536.226  mm,	Z =   -248.030  mm,
	W =  90.000 deg,	P =   0.000 deg,	R =   90.000 deg
};
P[1372]{
   GP1:
	UF : 0, UT : 6,		CONFIG : 'N U T, 0, 0, 0',
	X =  341.644  mm,	Y =   -535.802  mm,	Z =   -247.803  mm,
	W =  90.000 deg,	P =   0.000 deg,	R =   90.000 deg
};
P[1373]{
   GP1:
	UF : 0, UT : 6,		CONFIG : 'N U T, 0, 0, 0',
	X =  342.254  mm,	Y =   -535.312  mm,	Z =   -248.140  mm,
	W =  90.000 deg,	P =   0.000 deg,	R =   90.000 deg
};
P[1374]{
   GP1:
	UF : 0, UT : 6,		CONFIG : 'N U T, 0, 0, 0',
	X =  342.923  mm,	Y =   -534.936  mm,	Z =   -248.114  mm,
	W =  90.000 deg,	P =   0.000 deg,	R =   90.000 deg
};
P[1375]{
   GP1:
	UF : 0, UT : 6,		CONFIG : 'N U T, 0, 0, 0',
	X =  346.634  mm,	Y =   -532.787  mm,	Z =   -248.129  mm,
	W =  90.000 deg,	P =   0.000 deg,	R =   90.000 deg
};
P[1376]{
   GP1:
	UF : 0, UT : 6,		CONFIG : 'N U T, 0, 0, 0',
	X =  348.394  mm,	Y =   -531.902  mm,	Z =   -247.811  mm,
	W =  90.000 deg,	P =   0.000 deg,	R =   90.000 deg
};
P[1377]{
   GP1:
	UF : 0, UT : 6,		CONFIG : 'N U T, 0, 0, 0',
	X =  351.297  mm,	Y =   -530.232  mm,	Z =   -247.796  mm,
	W =  90.000 deg,	P =   0.000 deg,	R =   90.000 deg
};
P[1378]{
   GP1:
	UF : 0, UT : 6,		CONFIG : 'N U T, 0, 0, 0',
	X =  353.664  mm,	Y =   -528.843  mm,	Z =   -247.851  mm,
	W =  90.000 deg,	P =   0.000 deg,	R =   90.000 deg
};
P[1379]{
   GP1:
	UF : 0, UT : 6,		CONFIG : 'N U T, 0, 0, 0',
	X =  355.170  mm,	Y =   -527.882  mm,	Z =   -248.072  mm,
	W =  90.000 deg,	P =   0.000 deg,	R =   90.000 deg
};
P[1380]{
   GP1:
	UF : 0, UT : 6,		CONFIG : 'N U T, 0, 0, 0',
	X =  356.468  mm,	Y =   -527.061  mm,	Z =   -248.245  mm,
	W =  90.000 deg,	P =   0.000 deg,	R =   90.000 deg
};
P[1381]{
   GP1:
	UF : 0, UT : 6,		CONFIG : 'N U T, 0, 0, 0',
	X =  357.790  mm,	Y =   -526.488  mm,	Z =   -247.784  mm,
	W =  90.000 deg,	P =   0.000 deg,	R =   90.000 deg
};
P[1382]{
   GP1:
	UF : 0, UT : 6,		CONFIG : 'N U T, 0, 0, 0',
	X =  358.679  mm,	Y =   -525.886  mm,	Z =   -247.999  mm,
	W =  90.000 deg,	P =   0.000 deg,	R =   90.000 deg
};
P[1383]{
   GP1:
	UF : 0, UT : 6,		CONFIG : 'N U T, 0, 0, 0',
	X =  361.501  mm,	Y =   -524.298  mm,	Z =   -247.898  mm,
	W =  90.000 deg,	P =   0.000 deg,	R =   90.000 deg
};
P[1384]{
   GP1:
	UF : 0, UT : 6,		CONFIG : 'N U T, 0, 0, 0',
	X =  362.056  mm,	Y =   -523.868  mm,	Z =   -248.165  mm,
	W =  90.000 deg,	P =   0.000 deg,	R =   90.000 deg
};
P[1385]{
   GP1:
	UF : 0, UT : 6,		CONFIG : 'N U T, 0, 0, 0',
	X =  362.616  mm,	Y =   -523.512  mm,	Z =   -248.240  mm,
	W =  90.000 deg,	P =   0.000 deg,	R =   90.000 deg
};
P[1386]{
   GP1:
	UF : 0, UT : 6,		CONFIG : 'N U T, 0, 0, 0',
	X =  363.282  mm,	Y =   -523.267  mm,	Z =   -247.906  mm,
	W =  90.000 deg,	P =   0.000 deg,	R =   90.000 deg
};
P[1387]{
   GP1:
	UF : 0, UT : 6,		CONFIG : 'N U T, 0, 0, 0',
	X =  364.856  mm,	Y =   -522.370  mm,	Z =   -247.874  mm,
	W =  90.000 deg,	P =   0.000 deg,	R =   90.000 deg
};
P[1388]{
   GP1:
	UF : 0, UT : 6,		CONFIG : 'N U T, 0, 0, 0',
	X =  367.883  mm,	Y =   -520.631  mm,	Z =   -247.856  mm,
	W =  90.000 deg,	P =   0.000 deg,	R =   90.000 deg
};
P[1389]{
   GP1:
	UF : 0, UT : 6,		CONFIG : 'N U T, 0, 0, 0',
	X =  370.836  mm,	Y =   -518.859  mm,	Z =   -248.016  mm,
	W =  90.000 deg,	P =   0.000 deg,	R =   90.000 deg
};
P[1390]{
   GP1:
	UF : 0, UT : 6,		CONFIG : 'N U T, 0, 0, 0',
	X =  373.653  mm,	Y =   -517.291  mm,	Z =   -247.874  mm,
	W =  90.000 deg,	P =   0.000 deg,	R =   90.000 deg
};
P[1391]{
   GP1:
	UF : 0, UT : 6,		CONFIG : 'N U T, 0, 0, 0',
	X =  377.774  mm,	Y =   -514.851  mm,	Z =   -248.023  mm,
	W =  90.000 deg,	P =   0.000 deg,	R =   90.000 deg
};
P[1392]{
   GP1:
	UF : 0, UT : 6,		CONFIG : 'N U T, 0, 0, 0',
	X =  379.154  mm,	Y =   -513.985  mm,	Z =   -248.191  mm,
	W =  90.000 deg,	P =   0.000 deg,	R =   90.000 deg
};
P[1393]{
   GP1:
	UF : 0, UT : 6,		CONFIG : 'N U T, 0, 0, 0',
	X =  379.765  mm,	Y =   -513.697  mm,	Z =   -248.035  mm,
	W =  90.000 deg,	P =   0.000 deg,	R =   90.000 deg
};
P[1394]{
   GP1:
	UF : 0, UT : 6,		CONFIG : 'N U T, 0, 0, 0',
	X =  380.353  mm,	Y =   -513.328  mm,	Z =   -248.104  mm,
	W =  90.000 deg,	P =   0.000 deg,	R =   90.000 deg
};
P[1395]{
   GP1:
	UF : 0, UT : 6,		CONFIG : 'N U T, 0, 0, 0',
	X =  381.474  mm,	Y =   -512.801  mm,	Z =   -247.812  mm,
	W =  90.000 deg,	P =   0.000 deg,	R =   90.000 deg
};
P[1396]{
   GP1:
	UF : 0, UT : 6,		CONFIG : 'N U T, 0, 0, 0',
	X =  382.451  mm,	Y =   -512.099  mm,	Z =   -248.150  mm,
	W =  90.000 deg,	P =   0.000 deg,	R =   90.000 deg
};
P[1397]{
   GP1:
	UF : 0, UT : 6,		CONFIG : 'N U T, 0, 0, 0',
	X =  383.221  mm,	Y =   -511.718  mm,	Z =   -247.992  mm,
	W =  90.000 deg,	P =   0.000 deg,	R =   90.000 deg
};
P[1398]{
   GP1:
	UF : 0, UT : 6,		CONFIG : 'N U T, 0, 0, 0',
	X =  383.794  mm,	Y =   -511.326  mm,	Z =   -248.142  mm,
	W =  90.000 deg,	P =   0.000 deg,	R =   90.000 deg
};
P[1399]{
   GP1:
	UF : 0, UT : 6,		CONFIG : 'N U T, 0, 0, 0',
	X =  384.784  mm,	Y =   -510.825  mm,	Z =   -247.969  mm,
	W =  90.000 deg,	P =   0.000 deg,	R =   90.000 deg
};
P[1400]{
   GP1:
	UF : 0, UT : 6,		CONFIG : 'N U T, 0, 0, 0',
	X =  387.283  mm,	Y =   -509.319  mm,	Z =   -248.125  mm,
	W =  90.000 deg,	P =   0.000 deg,	R =   90.000 deg
};
P[1401]{
   GP1:
	UF : 0, UT : 6,		CONFIG : 'N U T, 0, 0, 0',
	X =  388.539  mm,	Y =   -508.676  mm,	Z =   -247.922  mm,
	W =  90.000 deg,	P =   0.000 deg,	R =   90.000 deg
};
P[1402]{
   GP1:
	UF : 0, UT : 6,		CONFIG : 'N U T, 0, 0, 0',
	X =  389.937  mm,	Y =   -507.743  mm,	Z =   -248.228  mm,
	W =  90.000 deg,	P =   0.000 deg,	R =   90.000 deg
};
P[1403]{
   GP1:
	UF : 0, UT : 6,		CONFIG : 'N U T, 0, 0, 0',
	X =  390.649  mm,	Y =   -507.518  mm,	Z =   -247.780  mm,
	W =  90.000 deg,	P =   0.000 deg,	R =   90.000 deg
};
P[1404]{
   GP1:
	UF : 0, UT : 6,		CONFIG : 'N U T, 0, 0, 0',
	X =  391.516  mm,	Y =   -506.948  mm,	Z =   -247.945  mm,
	W =  90.000 deg,	P =   0.000 deg,	R =   90.000 deg
};
P[1405]{
   GP1:
	UF : 0, UT : 6,		CONFIG : 'N U T, 0, 0, 0',
	X =  392.576  mm,	Y =   -506.282  mm,	Z =   -248.077  mm,
	W =  90.000 deg,	P =   0.000 deg,	R =   90.000 deg
};
P[1406]{
   GP1:
	UF : 0, UT : 6,		CONFIG : 'N U T, 0, 0, 0',
	X =  393.347  mm,	Y =   -505.799  mm,	Z =   -248.167  mm,
	W =  90.000 deg,	P =   0.000 deg,	R =   90.000 deg
};
P[1407]{
   GP1:
	UF : 0, UT : 6,		CONFIG : 'N U T, 0, 0, 0',
	X =  394.011  mm,	Y =   -505.563  mm,	Z =   -247.812  mm,
	W =  90.000 deg,	P =   0.000 deg,	R =   90.000 deg
};
P[1408]{
   GP1:
	UF : 0, UT : 6,		CONFIG : 'N U T, 0, 0, 0',
	X =  395.400  mm,	Y =   -504.742  mm,	Z =   -247.856  mm,
	W =  90.000 deg,	P =   0.000 deg,	R =   90.000 deg
};
P[1409]{
   GP1:
	UF : 0, UT : 6,		CONFIG : 'N U T, 0, 0, 0',
	X =  397.594  mm,	Y =   -503.321  mm,	Z =   -248.231  mm,
	W =  90.000 deg,	P =   0.000 deg,	R =   90.000 deg
};
P[1410]{
   GP1:
	UF : 0, UT : 6,		CONFIG : 'N U T, 0, 0, 0',
	X =  399.946  mm,	Y =   -501.999  mm,	Z =   -248.143  mm,
	W =  90.000 deg,	P =   0.000 deg,	R =   90.000 deg
};
P[1411]{
   GP1:
	UF : 0, UT : 6,		CONFIG : 'N U T, 0, 0, 0',
	X =  401.991  mm,	Y =   -500.774  mm,	Z =   -248.251  mm,
	W =  90.000 deg,	P =   0.000 deg,	R =   90.000 deg
};
P[1412]{
   GP1:
	UF : 0, UT : 6,		CONFIG : 'N U T, 0, 0, 0',
	X =  402.770  mm,	Y =   -500.346  mm,	Z =   -248.198  mm,
	W =  90.000 deg,	P =   0.000 deg,	R =   90.000 deg
};
P[1413]{
   GP1:
	UF : 0, UT : 6,		CONFIG : 'N U T, 0, 0, 0',
	X =  403.799  mm,	Y =   -499.784  mm,	Z =   -248.122  mm,
	W =  90.000 deg,	P =   0.000 deg,	R =   90.000 deg
};
P[1414]{
   GP1:
	UF : 0, UT : 6,		CONFIG : 'N U T, 0, 0, 0',
	X =  404.998  mm,	Y =   -499.104  mm,	Z =   -248.092  mm,
	W =  90.000 deg,	P =   0.000 deg,	R =   90.000 deg
};
P[1415]{
   GP1:
	UF : 0, UT : 6,		CONFIG : 'N U T, 0, 0, 0',
	X =  407.234  mm,	Y =   -497.781  mm,	Z =   -248.167  mm,
	W =  90.000 deg,	P =   0.000 deg,	R =   90.000 deg
};
P[1416]{
   GP1:
	UF : 0, UT : 6,		CONFIG : 'N U T, 0, 0, 0',
	X =  410.163  mm,	Y =   -496.169  mm,	Z =   -247.976  mm,
	W =  90.000 deg,	P =   0.000 deg,	R =   90.000 deg
};
P[1417]{
   GP1:
	UF : 0, UT : 6,		CONFIG : 'N U T, 0, 0, 0',
	X =  410.902  mm,	Y =   -495.767  mm,	Z =   -247.916  mm,
	W =  90.000 deg,	P =   0.000 deg,	R =   90.000 deg
};
P[1418]{
   GP1:
	UF : 0, UT : 6,		CONFIG : 'N U T, 0, 0, 0',
	X =  411.977  mm,	Y =   -495.078  mm,	Z =   -248.080  mm,
	W =  90.000 deg,	P =   0.000 deg,	R =   90.000 deg
};
P[1419]{
   GP1:
	UF : 0, UT : 6,		CONFIG : 'N U T, 0, 0, 0',
	X =  415.471  mm,	Y =   -493.037  mm,	Z =   -248.139  mm,
	W =  90.000 deg,	P =   0.000 deg,	R =   90.000 deg
};
P[1420]{
   GP1:
	UF : 0, UT : 6,		CONFIG : 'N U T, 0, 0, 0',
	X =  417.288  mm,	Y =   -491.993  mm,	Z =   -248.128  mm,
	W =  90.000 deg,	P =   0.000 deg,	R =   90.000 deg
};
P[1421]{
   GP1:
	UF : 0, UT : 6,		CONFIG : 'N U T, 0, 0, 0',
	X =  418.285  mm,	Y =   -491.532  mm,	Z =   -247.848  mm,
	W =  90.000 deg,	P =   0.000 deg,	R =   90.000 deg
};
P[1422]{
   GP1:
	UF : 0, UT : 6,		CONFIG : 'N U T, 0, 0, 0',
	X =  422.182  mm,	Y =   -489.156  mm,	Z =   -248.155  mm,
	W =  90.000 deg,	P =   0.000 deg,	R =   90.000 deg
};
P[1423]{
   GP1:
	UF : 0, UT : 6,		CONFIG : 'N U T, 0, 0, 0',
	X =  422.926  mm,	Y =   -488.724  mm,	Z =   -248.159  mm,
	W =  90.000 deg,	P =   0.000 deg,	R =   90.000 deg
};
P[1424]{
   GP1:
	UF : 0, UT : 6,		CONFIG : 'N U T, 0, 0, 0',
	X =  424.269  mm,	Y =   -487.929  mm,	Z =   -248.207  mm,
	W =  90.000 deg,	P =   0.000 deg,	R =   90.000 deg
};
P[1425]{
   GP1:
	UF : 0, UT : 6,		CONFIG : 'N U T, 0, 0, 0',
	X =  426.128  mm,	Y =   -486.979  mm,	Z =   -247.908  mm,
	W =  90.000 deg,	P =   0.000 deg,	R =   90.000 deg
};
P[1426]{
   GP1:
	UF : 0, UT : 6,		CONFIG : 'N U T, 0, 0, 0',
	X =  426.912  mm,	Y =   -486.484  mm,	Z =   -248.010  mm,
	W =  90.000 deg,	P =   0.000 deg,	R =   90.000 deg
};
P[1427]{
   GP1:
	UF : 0, UT : 6,		CONFIG : 'N U T, 0, 0, 0',
	X =  427.912  mm,	Y =   -485.890  mm,	Z =   -248.050  mm,
	W =  90.000 deg,	P =   0.000 deg,	R =   90.000 deg
};
P[1428]{
   GP1:
	UF : 0, UT : 6,		CONFIG : 'N U T, 0, 0, 0',
	X =  429.376  mm,	Y =   -484.988  mm,	Z =   -248.189  mm,
	W =  90.000 deg,	P =   0.000 deg,	R =   90.000 deg
};
P[1429]{
   GP1:
	UF : 0, UT : 6,		CONFIG : 'N U T, 0, 0, 0',
	X =  431.864  mm,	Y =   -483.549  mm,	Z =   -248.194  mm,
	W =  90.000 deg,	P =   0.000 deg,	R =   90.000 deg
};
P[1430]{
   GP1:
	UF : 0, UT : 6,		CONFIG : 'N U T, 0, 0, 0',
	X =  433.066  mm,	Y =   -482.906  mm,	Z =   -248.070  mm,
	W =  90.000 deg,	P =   0.000 deg,	R =   90.000 deg
};
P[1431]{
   GP1:
	UF : 0, UT : 6,		CONFIG : 'N U T, 0, 0, 0',
	X =  434.325  mm,	Y =   -482.187  mm,	Z =   -248.053  mm,
	W =  90.000 deg,	P =   0.000 deg,	R =   90.000 deg
};
P[1432]{
   GP1:
	UF : 0, UT : 6,		CONFIG : 'N U T, 0, 0, 0',
	X =  437.277  mm,	Y =   -480.444  mm,	Z =   -248.143  mm,
	W =  90.000 deg,	P =   0.000 deg,	R =   90.000 deg
};
P[1433]{
   GP1:
	UF : 0, UT : 6,		CONFIG : 'N U T, 0, 0, 0',
	X =  438.752  mm,	Y =   -479.580  mm,	Z =   -248.173  mm,
	W =  90.000 deg,	P =   0.000 deg,	R =   90.000 deg
};
P[1434]{
   GP1:
	UF : 0, UT : 6,		CONFIG : 'N U T, 0, 0, 0',
	X =  439.647  mm,	Y =   -479.087  mm,	Z =   -248.115  mm,
	W =  90.000 deg,	P =   0.000 deg,	R =   90.000 deg
};
P[1435]{
   GP1:
	UF : 0, UT : 6,		CONFIG : 'N U T, 0, 0, 0',
	X =  440.842  mm,	Y =   -478.377  mm,	Z =   -248.165  mm,
	W =  90.000 deg,	P =   0.000 deg,	R =   90.000 deg
};
P[1436]{
   GP1:
	UF : 0, UT : 6,		CONFIG : 'N U T, 0, 0, 0',
	X =  442.545  mm,	Y =   -477.491  mm,	Z =   -247.930  mm,
	W =  90.000 deg,	P =   0.000 deg,	R =   90.000 deg
};
P[1437]{
   GP1:
	UF : 0, UT : 6,		CONFIG : 'N U T, 0, 0, 0',
	X =  444.797  mm,	Y =   -476.207  mm,	Z =   -247.891  mm,
	W =  90.000 deg,	P =   0.000 deg,	R =   90.000 deg
};
P[1438]{
   GP1:
	UF : 0, UT : 6,		CONFIG : 'N U T, 0, 0, 0',
	X =  449.959  mm,	Y =   -473.079  mm,	Z =   -248.246  mm,
	W =  90.000 deg,	P =   0.000 deg,	R =   90.000 deg
};
P[1439]{
   GP1:
	UF : 0, UT : 6,		CONFIG : 'N U T, 0, 0, 0',
	X =  450.650  mm,	Y =   -472.776  mm,	Z =   -248.015  mm,
	W =  90.000 deg,	P =   0.000 deg,	R =   90.000 deg
};
P[1440]{
   GP1:
	UF : 0, UT : 6,		CONFIG : 'N U T, 0, 0, 0',
	X =  451.629  mm,	Y =   -472.135  mm,	Z =   -248.198  mm,
	W =  90.000 deg,	P =   0.000 deg,	R =   90.000 deg
};
P[1441]{
   GP1:
	UF : 0, UT : 6,		CONFIG : 'N U T, 0, 0, 0',
	X =  454.117  mm,	Y =   -470.701  mm,	Z =   -248.191  mm,
	W =  90.000 deg,	P =   0.000 deg,	R =   90.000 deg
};
P[1442]{
   GP1:
	UF : 0, UT : 6,		CONFIG : 'N U T, 0, 0, 0',
	X =  457.624  mm,	Y =   -468.672  mm,	Z =   -248.201  mm,
	W =  90.000 deg,	P =   0.000 deg,	R =   90.000 deg
};
P[1443]{
   GP1:
	UF : 0, UT : 6,		CONFIG : 'N U T, 0, 0, 0',
	X =  459.526  mm,	Y =   -467.605  mm,	Z =   -248.127  mm,
	W =  90.000 deg,	P =   0.000 deg,	R =   90.000 deg
};
P[1444]{
   GP1:
	UF : 0, UT : 6,		CONFIG : 'N U T, 0, 0, 0',
	X =  464.797  mm,	Y =   -464.576  mm,	Z =   -248.090  mm,
	W =  90.000 deg,	P =   0.000 deg,	R =   90.000 deg
};
P[1445]{
   GP1:
	UF : 0, UT : 6,		CONFIG : 'N U T, 0, 0, 0',
	X =  465.655  mm,	Y =   -464.090  mm,	Z =   -248.070  mm,
	W =  90.000 deg,	P =   0.000 deg,	R =   90.000 deg
};
P[1446]{
   GP1:
	UF : 0, UT : 6,		CONFIG : 'N U T, 0, 0, 0',
	X =  468.734  mm,	Y =   -462.280  mm,	Z =   -248.147  mm,
	W =  90.000 deg,	P =   0.000 deg,	R =   90.000 deg
};
P[1447]{
   GP1:
	UF : 0, UT : 6,		CONFIG : 'N U T, 0, 0, 0',
	X =  469.903  mm,	Y =   -461.714  mm,	Z =   -247.883  mm,
	W =  90.000 deg,	P =   0.000 deg,	R =   90.000 deg
};
P[1448]{
   GP1:
	UF : 0, UT : 6,		CONFIG : 'N U T, 0, 0, 0',
	X =  470.506  mm,	Y =   -461.355  mm,	Z =   -247.909  mm,
	W =  90.000 deg,	P =   0.000 deg,	R =   90.000 deg
};
P[1449]{
   GP1:
	UF : 0, UT : 6,		CONFIG : 'N U T, 0, 0, 0',
	X =  472.113  mm,	Y =   -460.351  mm,	Z =   -248.095  mm,
	W =  90.000 deg,	P =   0.000 deg,	R =   90.000 deg
};
P[1450]{
   GP1:
	UF : 0, UT : 6,		CONFIG : 'N U T, 0, 0, 0',
	X =  474.070  mm,	Y =   -459.224  mm,	Z =   -248.087  mm,
	W =  90.000 deg,	P =   0.000 deg,	R =   90.000 deg
};
P[1451]{
   GP1:
	UF : 0, UT : 6,		CONFIG : 'N U T, 0, 0, 0',
	X =  476.520  mm,	Y =   -457.871  mm,	Z =   -247.938  mm,
	W =  90.000 deg,	P =   0.000 deg,	R =   90.000 deg
};
P[1452]{
   GP1:
	UF : 0, UT : 6,		CONFIG : 'N U T, 0, 0, 0',
	X =  477.065  mm,	Y =   -457.430  mm,	Z =   -248.242  mm,
	W =  90.000 deg,	P =   0.000 deg,	R =   90.000 deg
};
P[1453]{
   GP1:
	UF : 0, UT : 6,		CONFIG : 'N U T, 0, 0, 0',
	X =  477.930  mm,	Y =   -456.963  mm,	Z =   -248.164  mm,
	W =  90.000 deg,	P =   0.000 deg,	R =   90.000 deg
};
P[1454]{
   GP1:
	UF : 0, UT : 6,		CONFIG : 'N U T, 0, 0, 0',
	X =  478.953  mm,	Y =   -456.458  mm,	Z =   -247.956  mm,
	W =  90.000 deg,	P =   0.000 deg,	R =   90.000 deg
};
P[1455]{
   GP1:
	UF : 0, UT : 6,		CONFIG : 'N U T, 0, 0, 0',
	X =  479.833  mm,	Y =   -455.898  mm,	Z =   -248.082  mm,
	W =  90.000 deg,	P =   0.000 deg,	R =   90.000 deg
};
P[1456]{
   GP1:
	UF : 0, UT : 6,		CONFIG : 'N U T, 0, 0, 0',
	X =  480.972  mm,	Y =   -455.251  mm,	Z =   -248.056  mm,
	W =  90.000 deg,	P =   0.000 deg,	R =   90.000 deg
};
P[1457]{
   GP1:
	UF : 0, UT : 6,		CONFIG : 'N U T, 0, 0, 0',
	X =  481.524  mm,	Y =   -454.854  mm,	Z =   -248.248  mm,
	W =  90.000 deg,	P =   0.000 deg,	R =   90.000 deg
};
P[1458]{
   GP1:
	UF : 0, UT : 6,		CONFIG : 'N U T, 0, 0, 0',
	X =  483.316  mm,	Y =   -454.014  mm,	Z =   -247.775  mm,
	W =  90.000 deg,	P =   0.000 deg,	R =   90.000 deg
};
P[1459]{
   GP1:
	UF : 0, UT : 6,		CONFIG : 'N U T, 0, 0, 0',
	X =  483.890  mm,	Y =   -453.596  mm,	Z =   -247.985  mm,
	W =  90.000 deg,	P =   0.000 deg,	R =   90.000 deg
};
P[1460]{
   GP1:
	UF : 0, UT : 6,		CONFIG : 'N U T, 0, 0, 0',
	X =  485.297  mm,	Y =   -452.713  mm,	Z =   -248.158  mm,
	W =  90.000 deg,	P =   0.000 deg,	R =   90.000 deg
};
P[1461]{
   GP1:
	UF : 0, UT : 6,		CONFIG : 'N U T, 0, 0, 0',
	X =  486.964  mm,	Y =   -451.831  mm,	Z =   -247.963  mm,
	W =  90.000 deg,	P =   0.000 deg,	R =   90.000 deg
};
P[1462]{
   GP1:
	UF : 0, UT : 6,		CONFIG : 'N U T, 0, 0, 0',
	X =  488.511  mm,	Y =   -450.982  mm,	Z =   -247.852  mm,
	W =  90.000 deg,	P =   0.000 deg,	R =   90.000 deg
};
P[1463]{
   GP1:
	UF : 0, UT : 6,		CONFIG : 'N U T, 0, 0, 0',
	X =  489.903  mm,	Y =   -450.169  mm,	Z =   -247.878  mm,
	W =  90.000 deg,	P =   0.000 deg,	R =   90.000 deg
};
P[1464]{
   GP1:
	UF : 0, UT : 6,		CONFIG : 'N U T, 0, 0, 0',
	X =  490.487  mm,	Y =   -449.708  mm,	Z =   -248.176  mm,
	W =  90.000 deg,	P =   0.000 deg,	R =   90.000 deg
};
P[1465]{
   GP1:
	UF : 0, UT : 6,		CONFIG : 'N U T, 0, 0, 0',
	X =  492.425  mm,	Y =   -448.719  mm,	Z =   -247.861  mm,
	W =  90.000 deg,	P =   0.000 deg,	R =   90.000 deg
};
P[1466]{
   GP1:
	UF : 0, UT : 6,		CONFIG : 'N U T, 0, 0, 0',
	X =  494.068  mm,	Y =   -447.644  mm,	Z =   -248.168  mm,
	W =  90.000 deg,	P =   0.000 deg,	R =   90.000 deg
};
P[1467]{
   GP1:
	UF : 0, UT : 6,		CONFIG : 'N U T, 0, 0, 0',
	X =  494.894  mm,	Y =   -447.302  mm,	Z =   -247.839  mm,
	W =  90.000 deg,	P =   0.000 deg,	R =   90.000 deg
};
P[1468]{
   GP1:
	UF : 0, UT : 6,		CONFIG : 'N U T, 0, 0, 0',
	X =  495.465  mm,	Y =   -446.833  mm,	Z =   -248.178  mm,
	W =  90.000 deg,	P =   0.000 deg,	R =   90.000 deg
};
P[1469]{
   GP1:
	UF : 0, UT : 6,		CONFIG : 'N U T, 0, 0, 0',
	X =  498.523  mm,	Y =   -445.112  mm,	Z =   -248.068  mm,
	W =  90.000 deg,	P =   0.000 deg,	R =   90.000 deg
};
P[1470]{
   GP1:
	UF : 0, UT : 6,		CONFIG : 'N U T, 0, 0, 0',
	X =  499.928  mm,	Y =   -444.282  mm,	Z =   -248.115  mm,
	W =  90.000 deg,	P =   0.000 deg,	R =   90.000 deg
};
P[1471]{
   GP1:
	UF : 0, UT : 6,		CONFIG : 'N U T, 0, 0, 0',
	X =  501.712  mm,	Y =   -443.247  mm,	Z =   -248.127  mm,
	W =  90.000 deg,	P =   0.000 deg,	R =   90.000 deg
};
P[1472]{
   GP1:
	UF : 0, UT : 6,		CONFIG : 'N U T, 0, 0, 0',
	X =  502.765  mm,	Y =   -442.737  mm,	Z =   -247.892  mm,
	W =  90.000 deg,	P =   0.000 deg,	R =   90.000 deg
};
P[1473]{
   GP1:
	UF : 0, UT : 6,		CONFIG : 'N U T, 0, 0, 0',
	X =  508.198  mm,	Y =   -439.602  mm,	Z =   -247.885  mm,
	W =  90.000 deg,	P =   0.000 deg,	R =   90.000 deg
};
P[1474]{
   GP1:
	UF : 0, UT : 6,		CONFIG : 'N U T, 0, 0, 0',
	X =  511.641  mm,	Y =   -437.551  mm,	Z =   -248.041  mm,
	W =  90.000 deg,	P =   0.000 deg,	R =   90.000 deg
};
P[1475]{
   GP1:
	UF : 0, UT : 6,		CONFIG : 'N U T, 0, 0, 0',
	X =  513.759  mm,	Y =   -436.283  mm,	Z =   -248.145  mm,
	W =  90.000 deg,	P =   0.000 deg,	R =   90.000 deg
};
P[1476]{
   GP1:
	UF : 0, UT : 6,		CONFIG : 'N U T, 0, 0, 0',
	X =  514.369  mm,	Y =   -435.895  mm,	Z =   -248.233  mm,
	W =  90.000 deg,	P =   0.000 deg,	R =   90.000 deg
};
P[1477]{
   GP1:
	UF : 0, UT : 6,		CONFIG : 'N U T, 0, 0, 0',
	X =  515.120  mm,	Y =   -435.513  mm,	Z =   -248.106  mm,
	W =  90.000 deg,	P =   0.000 deg,	R =   90.000 deg
};
P[1478]{
   GP1:
	UF : 0, UT : 6,		CONFIG : 'N U T, 0, 0, 0',
	X =  515.898  mm,	Y =   -435.068  mm,	Z =   -248.099  mm,
	W =  90.000 deg,	P =   0.000 deg,	R =   90.000 deg
};
P[1479]{
   GP1:
	UF : 0, UT : 6,		CONFIG : 'N U T, 0, 0, 0',
	X =  516.874  mm,	Y =   -434.536  mm,	Z =   -247.962  mm,
	W =  90.000 deg,	P =   0.000 deg,	R =   90.000 deg
};
P[1480]{
   GP1:
	UF : 0, UT : 6,		CONFIG : 'N U T, 0, 0, 0',
	X =  519.453  mm,	Y =   -432.453  mm,	Z =   -248.155  mm,
	W =  90.000 deg,	P =   0.000 deg,	R =   90.000 deg
};
P[1481]{
   GP1:
	UF : 0, UT : 6,		CONFIG : 'N U T, 0, 0, 0',
	X =  520.384  mm,	Y =   -431.591  mm,	Z =   -247.897  mm,
	W =  90.000 deg,	P =   0.000 deg,	R =   90.000 deg
};
P[1482]{
   GP1:
	UF : 0, UT : 6,		CONFIG : 'N U T, 0, 0, 0',
	X =  521.918  mm,	Y =   -429.318  mm,	Z =   -248.035  mm,
	W =  90.000 deg,	P =   0.000 deg,	R =   90.000 deg
};
P[1483]{
   GP1:
	UF : 0, UT : 6,		CONFIG : 'N U T, 0, 0, 0',
	X =  522.512  mm,	Y =   -428.345  mm,	Z =   -247.911  mm,
	W =  90.000 deg,	P =   0.000 deg,	R =   90.000 deg
};
P[1484]{
   GP1:
	UF : 0, UT : 6,		CONFIG : 'N U T, 0, 0, 0',
	X =  523.273  mm,	Y =   -425.540  mm,	Z =   -248.190  mm,
	W =  90.000 deg,	P =   0.000 deg,	R =   90.000 deg
};
P[1485]{
   GP1:
	UF : 0, UT : 6,		CONFIG : 'N U T, 0, 0, 0',
	X =  523.492  mm,	Y =   -423.936  mm,	Z =   -248.204  mm,
	W =  90.000 deg,	P =   0.000 deg,	R =   90.000 deg
};
P[1486]{
   GP1:
	UF : 0, UT : 6,		CONFIG : 'N U T, 0, 0, 0',
	X =  521.137  mm,	Y =   -414.667  mm,	Z =   -247.874  mm,
	W =  90.000 deg,	P =   0.000 deg,	R =   90.000 deg
};
P[1487]{
   GP1:
	UF : 0, UT : 6,		CONFIG : 'N U T, 0, 0, 0',
	X =  519.949  mm,	Y =   -412.824  mm,	Z =   -248.177  mm,
	W =  90.000 deg,	P =   0.000 deg,	R =   90.000 deg
};
P[1488]{
   GP1:
	UF : 0, UT : 6,		CONFIG : 'N U T, 0, 0, 0',
	X =  519.713  mm,	Y =   -412.184  mm,	Z =   -247.852  mm,
	W =  90.000 deg,	P =   0.000 deg,	R =   90.000 deg
};
P[1489]{
   GP1:
	UF : 0, UT : 6,		CONFIG : 'N U T, 0, 0, 0',
	X =  518.014  mm,	Y =   -409.467  mm,	Z =   -248.169  mm,
	W =  90.000 deg,	P =   0.000 deg,	R =   90.000 deg
};
P[1490]{
   GP1:
	UF : 0, UT : 6,		CONFIG : 'N U T, 0, 0, 0',
	X =  517.541  mm,	Y =   -408.395  mm,	Z =   -247.814  mm,
	W =  90.000 deg,	P =   0.000 deg,	R =   90.000 deg
};
P[1491]{
   GP1:
	UF : 0, UT : 6,		CONFIG : 'N U T, 0, 0, 0',
	X =  517.010  mm,	Y =   -407.748  mm,	Z =   -248.195  mm,
	W =  90.000 deg,	P =   0.000 deg,	R =   90.000 deg
};
P[1492]{
   GP1:
	UF : 0, UT : 6,		CONFIG : 'N U T, 0, 0, 0',
	X =  515.552  mm,	Y =   -405.035  mm,	Z =   -247.933  mm,
	W =  90.000 deg,	P =   0.000 deg,	R =   90.000 deg
};
P[1493]{
   GP1:
	UF : 0, UT : 6,		CONFIG : 'N U T, 0, 0, 0',
	X =  514.590  mm,	Y =   -403.551  mm,	Z =   -248.189  mm,
	W =  90.000 deg,	P =   0.000 deg,	R =   90.000 deg
};
P[1494]{
   GP1:
	UF : 0, UT : 6,		CONFIG : 'N U T, 0, 0, 0',
	X =  513.251  mm,	Y =   -401.250  mm,	Z =   -248.213  mm,
	W =  90.000 deg,	P =   0.000 deg,	R =   90.000 deg
};
P[1495]{
   GP1:
	UF : 0, UT : 6,		CONFIG : 'N U T, 0, 0, 0',
	X =  510.119  mm,	Y =   -395.575  mm,	Z =   -247.860  mm,
	W =  90.000 deg,	P =   0.000 deg,	R =   90.000 deg
};
P[1496]{
   GP1:
	UF : 0, UT : 6,		CONFIG : 'N U T, 0, 0, 0',
	X =  509.202  mm,	Y =   -394.169  mm,	Z =   -248.117  mm,
	W =  90.000 deg,	P =   0.000 deg,	R =   90.000 deg
};
P[1497]{
   GP1:
	UF : 0, UT : 6,		CONFIG : 'N U T, 0, 0, 0',
	X =  508.621  mm,	Y =   -393.170  mm,	Z =   -248.127  mm,
	W =  90.000 deg,	P =   0.000 deg,	R =   90.000 deg
};
P[1498]{
   GP1:
	UF : 0, UT : 6,		CONFIG : 'N U T, 0, 0, 0',
	X =  507.688  mm,	Y =   -391.501  mm,	Z =   -248.054  mm,
	W =  90.000 deg,	P =   0.000 deg,	R =   90.000 deg
};
P[1499]{
   GP1:
	UF : 0, UT : 6,		CONFIG : 'N U T, 0, 0, 0',
	X =  506.452  mm,	Y =   -389.306  mm,	Z =   -247.975  mm,
	W =  90.000 deg,	P =   0.000 deg,	R =   90.000 deg
};
P[1500]{
   GP1:
	UF : 0, UT : 6,		CONFIG : 'N U T, 0, 0, 0',
	X =  505.317  mm,	Y =   -387.531  mm,	Z =   -248.242  mm,
	W =  90.000 deg,	P =   0.000 deg,	R =   90.000 deg
};
P[1501]{
   GP1:
	UF : 0, UT : 6,		CONFIG : 'N U T, 0, 0, 0',
	X =  504.798  mm,	Y =   -386.435  mm,	Z =   -247.968  mm,
	W =  90.000 deg,	P =   0.000 deg,	R =   90.000 deg
};
P[1502]{
   GP1:
	UF : 0, UT : 6,		CONFIG : 'N U T, 0, 0, 0',
	X =  503.162  mm,	Y =   -383.655  mm,	Z =   -248.042  mm,
	W =  90.000 deg,	P =   0.000 deg,	R =   90.000 deg
};
P[1503]{
   GP1:
	UF : 0, UT : 6,		CONFIG : 'N U T, 0, 0, 0',
	X =  502.724  mm,	Y =   -383.038  mm,	Z =   -248.239  mm,
	W =  90.000 deg,	P =   0.000 deg,	R =   90.000 deg
};
P[1504]{
   GP1:
	UF : 0, UT : 6,		CONFIG : 'N U T, 0, 0, 0',
	X =  502.245  mm,	Y =   -382.119  mm,	Z =   -248.117  mm,
	W =  90.000 deg,	P =   0.000 deg,	R =   90.000 deg
};
P[1505]{
   GP1:
	UF : 0, UT : 6,		CONFIG : 'N U T, 0, 0, 0',
	X =  501.837  mm,	Y =   -381.359  mm,	Z =   -248.043  mm,
	W =  90.000 deg,	P =   0.000 deg,	R =   90.000 deg
};
P[1506]{
   GP1:
	UF : 0, UT : 6,		CONFIG : 'N U T, 0, 0, 0',
	X =  500.466  mm,	Y =   -379.006  mm,	Z =   -248.069  mm,
	W =  90.000 deg,	P =   0.000 deg,	R =   90.000 deg
};
P[1507]{
   GP1:
	UF : 0, UT : 6,		CONFIG : 'N U T, 0, 0, 0',
	X =  499.611  mm,	Y =   -377.409  mm,	Z =   -247.907  mm,
	W =  90.000 deg,	P =   0.000 deg,	R =   90.000 deg
};
P[1508]{
   GP1:
	UF : 0, UT : 6,		CONFIG : 'N U T, 0, 0, 0',
	X =  498.909  mm,	Y =   -376.345  mm,	Z =   -248.120  mm,
	W =  90.000 deg,	P =   0.000 deg,	R =   90.000 deg
};
P[1509]{
   GP1:
	UF : 0, UT : 6,		CONFIG : 'N U T, 0, 0, 0',
	X =  497.043  mm,	Y =   -373.154  mm,	Z =   -248.180  mm,
	W =  90.000 deg,	P =   0.000 deg,	R =   90.000 deg
};
P[1510]{
   GP1:
	UF : 0, UT : 6,		CONFIG : 'N U T, 0, 0, 0',
	X =  494.318  mm,	Y =   -368.455  mm,	Z =   -248.207  mm,
	W =  90.000 deg,	P =   0.000 deg,	R =   90.000 deg
};
P[1511]{
   GP1:
	UF : 0, UT : 6,		CONFIG : 'N U T, 0, 0, 0',
	X =  493.597  mm,	Y =   -366.953  mm,	Z =   -247.854  mm,
	W =  90.000 deg,	P =   0.000 deg,	R =   90.000 deg
};
P[1512]{
   GP1:
	UF : 0, UT : 6,		CONFIG : 'N U T, 0, 0, 0',
	X =  492.592  mm,	Y =   -365.229  mm,	Z =   -247.875  mm,
	W =  90.000 deg,	P =   0.000 deg,	R =   90.000 deg
};
P[1513]{
   GP1:
	UF : 0, UT : 6,		CONFIG : 'N U T, 0, 0, 0',
	X =  490.044  mm,	Y =   -360.952  mm,	Z =   -248.065  mm,
	W =  90.000 deg,	P =   0.000 deg,	R =   90.000 deg
};
P[1514]{
   GP1:
	UF : 0, UT : 6,		CONFIG : 'N U T, 0, 0, 0',
	X =  488.603  mm,	Y =   -358.440  mm,	Z =   -248.042  mm,
	W =  90.000 deg,	P =   0.000 deg,	R =   90.000 deg
};
P[1515]{
   GP1:
	UF : 0, UT : 6,		CONFIG : 'N U T, 0, 0, 0',
	X =  487.314  mm,	Y =   -356.225  mm,	Z =   -248.067  mm,
	W =  90.000 deg,	P =   0.000 deg,	R =   90.000 deg
};
P[1516]{
   GP1:
	UF : 0, UT : 6,		CONFIG : 'N U T, 0, 0, 0',
	X =  486.026  mm,	Y =   -354.044  mm,	Z =   -248.139  mm,
	W =  90.000 deg,	P =   0.000 deg,	R =   90.000 deg
};
P[1517]{
   GP1:
	UF : 0, UT : 6,		CONFIG : 'N U T, 0, 0, 0',
	X =  482.746  mm,	Y =   -348.427  mm,	Z =   -248.228  mm,
	W =  90.000 deg,	P =   0.000 deg,	R =   90.000 deg
};
P[1518]{
   GP1:
	UF : 0, UT : 6,		CONFIG : 'N U T, 0, 0, 0',
	X =  481.705  mm,	Y =   -346.539  mm,	Z =   -248.106  mm,
	W =  90.000 deg,	P =   0.000 deg,	R =   90.000 deg
};
P[1519]{
   GP1:
	UF : 0, UT : 6,		CONFIG : 'N U T, 0, 0, 0',
	X =  481.114  mm,	Y =   -345.390  mm,	Z =   -247.933  mm,
	W =  90.000 deg,	P =   0.000 deg,	R =   90.000 deg
};
P[1520]{
   GP1:
	UF : 0, UT : 6,		CONFIG : 'N U T, 0, 0, 0',
	X =  480.454  mm,	Y =   -344.453  mm,	Z =   -248.220  mm,
	W =  90.000 deg,	P =   0.000 deg,	R =   90.000 deg
};
P[1521]{
   GP1:
	UF : 0, UT : 6,		CONFIG : 'N U T, 0, 0, 0',
	X =  479.864  mm,	Y =   -343.185  mm,	Z =   -247.875  mm,
	W =  90.000 deg,	P =   0.000 deg,	R =   90.000 deg
};
P[1522]{
   GP1:
	UF : 0, UT : 6,		CONFIG : 'N U T, 0, 0, 0',
	X =  478.938  mm,	Y =   -341.835  mm,	Z =   -248.232  mm,
	W =  90.000 deg,	P =   0.000 deg,	R =   90.000 deg
};
P[1523]{
   GP1:
	UF : 0, UT : 6,		CONFIG : 'N U T, 0, 0, 0',
	X =  478.393  mm,	Y =   -340.791  mm,	Z =   -248.090  mm,
	W =  90.000 deg,	P =   0.000 deg,	R =   90.000 deg
};
P[1524]{
   GP1:
	UF : 0, UT : 6,		CONFIG : 'N U T, 0, 0, 0',
	X =  477.695  mm,	Y =   -339.621  mm,	Z =   -248.143  mm,
	W =  90.000 deg,	P =   0.000 deg,	R =   90.000 deg
};
P[1525]{
   GP1:
	UF : 0, UT : 6,		CONFIG : 'N U T, 0, 0, 0',
	X =  476.913  mm,	Y =   -338.020  mm,	Z =   -247.798  mm,
	W =  90.000 deg,	P =   0.000 deg,	R =   90.000 deg
};
P[1526]{
   GP1:
	UF : 0, UT : 6,		CONFIG : 'N U T, 0, 0, 0',
	X =  476.245  mm,	Y =   -336.964  mm,	Z =   -247.941  mm,
	W =  90.000 deg,	P =   0.000 deg,	R =   90.000 deg
};
P[1527]{
   GP1:
	UF : 0, UT : 6,		CONFIG : 'N U T, 0, 0, 0',
	X =  475.810  mm,	Y =   -336.340  mm,	Z =   -248.122  mm,
	W =  90.000 deg,	P =   0.000 deg,	R =   90.000 deg
};
P[1528]{
   GP1:
